LIN {X 0,Y 257.975,Z 573.967,A -85,B 0,C 180,E1 -19198.916,E2 -19198.916} C_VEL
LIN {X 0,Y 261.69,Z 562.431,A -85,B 0,C 180,E1 -19200.904,E2 -19200.904} C_VEL
LIN {X 0,Y 265.113,Z 550.939,A -85,B 0,C 180,E1 -19202.465,E2 -19202.465} C_VEL
LIN {X 0,Y 268.237,Z 538.403,A -85,B 0,C 180,E1 -19203.83,E2 -19203.83} C_VEL
LIN {X 0,Y 271.089,Z 525.455,A -85,B 0,C 180,E1 -19204.886,E2 -19204.886} C_VEL
LIN {X 0,Y 273.137,Z 513.119,A -85,B 0,C 180,E1 -19205.657,E2 -19205.657} C_VEL
LIN {X 0,Y 274.903,Z 498.669,A -85,B 0,C 180,E1 -19206.281,E2 -19206.281} C_VEL
LIN {X 0,Y 276.815,Z 466.117,A -85,B 0,C 180,E1 -19207.149,E2 -19207.149} C_VEL
LIN {X 0,Y 279.015,Z 421.953,A -85,B 0,C 180,E1 -19208.302,E2 -19208.302} C_VEL
LIN {X 0,Y 278.053,Z 415.902,A -85,B 0,C 180,E1 -19208.716,E2 -19208.716} C_VEL
LIN {X 0,Y 271.984,Z 402.227,A -85,B 0,C 180,E1 -19210.518,E2 -19210.518} C_VEL
LIN {X 0,Y 265.036,Z 388.919,A -85,B 0,C 180,E1 -19212.665,E2 -19212.665} C_VEL
LIN {X 0,Y 258.695,Z 378.17,A -85,B 0,C 180,E1 -19214.774,E2 -19214.774} C_VEL
LIN {X 0,Y 255.82,Z 373.588,A -85,B 0,C 180,E1 -19215.796,E2 -19215.796} C_VEL
LIN {X 0,Y 252.154,Z 368.029,A -85,B 0,C 180,E1 -19217.157,E2 -19217.157} C_VEL
LIN {X 0,Y 248.387,Z 362.468,A -85,B 0,C 180,E1 -19218.642,E2 -19218.642} C_VEL
LIN {X 0,Y 245.206,Z 357.875,A -85,B 0,C 180,E1 -19219.976,E2 -19219.976} C_VEL
LIN {X 0,Y 244.693,Z 356.869,A -85,B 0,C 180,E1 -19220.278,E2 -19220.278} C_VEL
LIN {X 0,Y 242.615,Z 351.052,A -85,B 0,C 180,E1 -19224.2,E2 -19224.2} C_VEL
LIN {X 0,Y 242.003,Z 348.966,A -85,B 0,C 180,E1 -19225.759,E2 -19225.759} C_VEL
LIN {X 0,Y 242.032,Z 348.953,A -85,B 0,C 180,E1 -19230.586,E2 -19230.586} C_VEL
LIN {X 0,Y 242.062,Z 348.949,A -85,B 0,C 180,E1 -19234.182,E2 -19234.182} C_VEL
LIN {X 0,Y 242.047,Z 348.954,A -85,B 0,C 180,E1 -19238.296,E2 -19238.296} C_VEL
LIN {X 0,Y 242.157,Z 348.946,A -85,B 0,C 180,E1 -19243.277,E2 -19243.277} C_VEL
LIN {X 0,Y 242.18,Z 348.932,A -85,B 0,C 180,E1 -19248.279,E2 -19248.279} C_VEL
LIN {X 0,Y 242.428,Z 348.909,A -85,B 0,C 180,E1 -19251.665,E2 -19251.665} C_VEL
LIN {X 0,Y 242.237,Z 348.937,A -85,B 0,C 180,E1 -19255.006,E2 -19255.006} C_VEL
LIN {X 0,Y 242.615,Z 348.882,A -85,B 0,C 180,E1 -19258.339,E2 -19258.339} C_VEL
LIN {X 0,Y 242.611,Z 348.878,A -85,B 0,C 180,E1 -19261.659,E2 -19261.659} C_VEL
LIN {X 0,Y 242.388,Z 348.915,A -85,B 0,C 180,E1 -19266.66,E2 -19266.66} C_VEL
LIN {X 0,Y 242.258,Z 348.927,A -85,B 0,C 180,E1 -19270.023,E2 -19270.023} C_VEL
LIN {X 0,Y 242.118,Z 348.946,A -85,B 0,C 180,E1 -19275.143,E2 -19275.143} C_VEL
LIN {X 0,Y 242.033,Z 348.956,A -85,B 0,C 180,E1 -19278.627,E2 -19278.627} C_VEL
LIN {X 0,Y 242.051,Z 349.148,A -85,B 0,C 180,E1 -19280.941,E2 -19280.941} C_VEL
LIN {X 0,Y 242.928,Z 351.572,A -85,B 0,C 180,E1 -19281.413,E2 -19281.413} C_VEL
LIN {X 0,Y 244.626,Z 353.64,A -85,B 0,C 180,E1 -19282.152,E2 -19282.152} C_VEL
LIN {X 0,Y 246.198,Z 354.858,A -85,B 0,C 180,E1 -19282.777,E2 -19282.777} C_VEL
LIN {X 0,Y 247.972,Z 357.809,A -85,B 0,C 180,E1 -19283.543,E2 -19283.543} C_VEL
LIN {X 0,Y 250.246,Z 360.174,A -85,B 0,C 180,E1 -19284.416,E2 -19284.416} C_VEL
LIN {X 0,Y 252.657,Z 363.577,A -85,B 0,C 180,E1 -19285.344,E2 -19285.344} C_VEL
LIN {X 0,Y 254.065,Z 365.243,A -85,B 0,C 180,E1 -19285.854,E2 -19285.854} C_VEL
LIN {X 0,Y 257.823,Z 370.434,A -85,B 0,C 180,E1 -19287.194,E2 -19287.194} C_VEL
LIN {X 0,Y 263.731,Z 378.79,A -85,B 0,C 180,E1 -19289.154,E2 -19289.154} C_VEL
LIN {X 0,Y 268.187,Z 385.843,A -85,B 0,C 180,E1 -19290.532,E2 -19290.532} C_VEL
LIN {X 0,Y 274.772,Z 397.82,A -85,B 0,C 180,E1 -19292.488,E2 -19292.488} C_VEL
LIN {X 0,Y 279.803,Z 408.378,A -85,B 0,C 180,E1 -19293.928,E2 -19293.928} C_VEL
LIN {X 0,Y 275.706,Z 481.995,A -85,B 0,C 180,E1 -19295.821,E2 -19295.821} C_VEL
LIN {X 0,Y 274.177,Z 496.417,A -85,B 0,C 180,E1 -19296.459,E2 -19296.459} C_VEL
LIN {X 0,Y 271.973,Z 510.678,A -85,B 0,C 180,E1 -19297.385,E2 -19297.385} C_VEL
LIN {X 0,Y 269.519,Z 523.528,A -85,B 0,C 180,E1 -19298.533,E2 -19298.533} C_VEL
LIN {X 0,Y 266.589,Z 535.608,A -85,B 0,C 180,E1 -19299.895,E2 -19299.895} C_VEL
LIN {X 0,Y 263.53,Z 546.378,A -85,B 0,C 180,E1 -19301.407,E2 -19301.407} C_VEL
LIN {X 0,Y 259.867,Z 557.729,A -85,B 0,C 180,E1 -19303.382,E2 -19303.382} C_VEL
LIN {X 0,Y 256.225,Z 567.968,A -85,B 0,C 180,E1 -19305.616,E2 -19305.616} C_VEL
LIN {X 0,Y 252.654,Z 577.137,A -85,B 0,C 180,E1 -19308.12,E2 -19308.12} C_VEL
LIN {X 0,Y 249.548,Z 584.618,A -85,B 0,C 180,E1 -19310.681,E2 -19310.681} C_VEL
LIN {X 0,Y 246.917,Z 590.719,A -85,B 0,C 180,E1 -19313.295,E2 -19313.295} C_VEL
LIN {X 0,Y 244.315,Z 596.539,A -85,B 0,C 180,E1 -19316.533,E2 -19316.533} C_VEL
LIN {X 0,Y 242.516,Z 600.511,A -85,B 0,C 180,E1 -19319.528,E2 -19319.528} C_VEL
LIN {X 0,Y 241.298,Z 603.047,A -85,B 0,C 180,E1 -19322.226,E2 -19322.226} C_VEL
LIN {X 0,Y 240.472,Z 604.693,A -85,B 0,C 180,E1 -19324.957,E2 -19324.957} C_VEL
LIN {X 0,Y 239.921,Z 605.496,A -85,B 0,C 180,E1 -19327.618,E2 -19327.618} C_VEL
LIN {X 0,Y 239.591,Z 605.256,A -85,B 0,C 180,E1 -19331.178,E2 -19331.178} C_VEL
LIN {X 0,Y 239.637,Z 603.584,A -85,B 0,C 180,E1 -19334.697,E2 -19334.697} C_VEL
LIN {X 0,Y 240.013,Z 600.481,A -85,B 0,C 180,E1 -19338.174,E2 -19338.174} C_VEL
LIN {X 0,Y 240.569,Z 597.158,A -85,B 0,C 180,E1 -19340.755,E2 -19340.755} C_VEL
LIN {X 0,Y 241.354,Z 592.961,A -85,B 0,C 180,E1 -19343.313,E2 -19343.313} C_VEL
LIN {X 0,Y 242.308,Z 587.757,A -85,B 0,C 180,E1 -19345.843,E2 -19345.843} C_VEL
LIN {X 0,Y 243.892,Z 580.311,A -85,B 0,C 180,E1 -19348.763,E2 -19348.763} C_VEL
LIN {X 0,Y 245.618,Z 572.504,A -85,B 0,C 180,E1 -19351.231,E2 -19351.231} C_VEL
LIN {X 0,Y 247.632,Z 563.136,A -85,B 0,C 180,E1 -19353.663,E2 -19353.663} C_VEL
LIN {X 0,Y 249.825,Z 552.746,A -85,B 0,C 180,E1 -19355.854,E2 -19355.854} C_VEL
LIN {X 0,Y 252.095,Z 541.274,A -85,B 0,C 180,E1 -19357.812,E2 -19357.812} C_VEL
LIN {X 0,Y 254.36,Z 528.566,A -85,B 0,C 180,E1 -19359.544,E2 -19359.544} C_VEL
LIN {X 0,Y 256.247,Z 516.233,A -85,B 0,C 180,E1 -19360.87,E2 -19360.87} C_VEL
LIN {X 0,Y 257.878,Z 502.651,A -85,B 0,C 180,E1 -19361.995,E2 -19361.995} C_VEL
LIN {X 0,Y 259.068,Z 489.521,A -85,B 0,C 180,E1 -19362.785,E2 -19362.785} C_VEL
LIN {X 0,Y 259.965,Z 475.474,A -85,B 0,C 180,E1 -19363.334,E2 -19363.334} C_VEL
LIN {X 0,Y 263.004,Z 394.213,A -85,B 0,C 180,E1 -19365.519,E2 -19365.519} C_VEL
LIN {X 0,Y 255.473,Z 375.166,A -85,B 0,C 180,E1 -19367.04,E2 -19367.04} C_VEL
LIN {X 0,Y 248.343,Z 361.226,A -85,B 0,C 180,E1 -19368.445,E2 -19368.445} C_VEL
LIN {X 0,Y 243.171,Z 351.999,A -85,B 0,C 180,E1 -19369.494,E2 -19369.494} C_VEL
LIN {X 0,Y 242.129,Z 349.364,A -85,B 0,C 180,E1 -19369.74,E2 -19369.74} C_VEL
LIN {X 0,Y 242.068,Z 348.964,A -85,B 0,C 180,E1 -19369.773,E2 -19369.773} C_VEL
LIN {X 0,Y 242.024,Z 348.964,A -85,B 0,C 180,E1 -19373.989,E2 -19373.989} C_VEL
LIN {X 0,Y 241.96,Z 348.97,A -85,B 0,C 180,E1 -19377.695,E2 -19377.695} C_VEL
LIN {X 0,Y 241.948,Z 348.97,A -85,B 0,C 180,E1 -19381.525,E2 -19381.525} C_VEL
LIN {X 0,Y 241.978,Z 348.959,A -85,B 0,C 180,E1 -19385.589,E2 -19385.589} C_VEL
LIN {X 0,Y 241.94,Z 348.972,A -85,B 0,C 180,E1 -19389.724,E2 -19389.724} C_VEL
LIN {X 0,Y 241.897,Z 348.958,A -85,B 0,C 180,E1 -19394.212,E2 -19394.212} C_VEL
LIN {X 0,Y 241.906,Z 348.974,A -85,B 0,C 180,E1 -19398.072,E2 -19398.072} C_VEL
LIN {X 0,Y 241.966,Z 348.95,A -85,B 0,C 180,E1 -19402.415,E2 -19402.415} C_VEL
LIN {X 0,Y 241.98,Z 348.956,A -85,B 0,C 180,E1 -19406.508,E2 -19406.508} C_VEL
LIN {X 0,Y 241.973,Z 348.967,A -85,B 0,C 180,E1 -19410.617,E2 -19410.617} C_VEL
LIN {X 0,Y 241.998,Z 348.964,A -85,B 0,C 180,E1 -19414.198,E2 -19414.198} C_VEL
LIN {X 0,Y 241.988,Z 348.961,A -85,B 0,C 180,E1 -19418.339,E2 -19418.339} C_VEL
LIN {X 0,Y 242.109,Z 348.947,A -85,B 0,C 180,E1 -19423.325,E2 -19423.325} C_VEL
LIN {X 0,Y 242.157,Z 348.916,A -85,B 0,C 180,E1 -19428.279,E2 -19428.279} C_VEL
LIN {X 0,Y 242.372,Z 348.913,A -85,B 0,C 180,E1 -19431.664,E2 -19431.664} C_VEL
LIN {X 0,Y 242.402,Z 348.913,A -85,B 0,C 180,E1 -19433.341,E2 -19433.341} C_VEL
LIN {X 0,Y 242.629,Z 348.862,A -85,B 0,C 180,E1 -19438.341,E2 -19438.341} C_VEL
LIN {X 0,Y 242.628,Z 348.869,A -85,B 0,C 180,E1 -19441.66,E2 -19441.66} C_VEL
LIN {X 0,Y 242.412,Z 348.911,A -85,B 0,C 180,E1 -19446.66,E2 -19446.66} C_VEL
LIN {X 0,Y 242.38,Z 348.91,A -85,B 0,C 180,E1 -19447.995,E2 -19447.995} C_VEL
LIN {X 0,Y 242.071,Z 348.952,A -85,B 0,C 180,E1 -19448.921,E2 -19448.921} C_VEL
LIN {X 0,Y 240.681,Z 349.13,A -85,B 0,C 180,E1 -19450.286,E2 -19450.286} C_VEL
LIN {X 0,Y 236.209,Z 349.682,A -85,B 0,C 180,E1 -19453.469,E2 -19453.469} C_VEL
LIN {X 0,Y 235.168,Z 349.812,A -85,B 0,C 180,E1 -19454.899,E2 -19454.899} C_VEL
LIN {X 0,Y 235.106,Z 349.821,A -85,B 0,C 180,E1 -19455.383,E2 -19455.383} C_VEL
LIN {X 0,Y 235.015,Z 349.828,A -85,B 0,C 180,E1 -19459.206,E2 -19459.206} C_VEL
LIN {X 0,Y 234.968,Z 349.839,A -85,B 0,C 180,E1 -19462.883,E2 -19462.883} C_VEL
LIN {X 0,Y 234.974,Z 349.837,A -85,B 0,C 180,E1 -19466.657,E2 -19466.657} C_VEL
LIN {X 0,Y 234.928,Z 349.842,A -85,B 0,C 180,E1 -19470.569,E2 -19470.569} C_VEL
LIN {X 0,Y 234.936,Z 349.844,A -85,B 0,C 180,E1 -19474.638,E2 -19474.638} C_VEL
LIN {X 0,Y 234.947,Z 349.833,A -85,B 0,C 180,E1 -19478.944,E2 -19478.944} C_VEL
LIN {X 0,Y 234.895,Z 349.851,A -85,B 0,C 180,E1 -19483.485,E2 -19483.485} C_VEL
LIN {X 0,Y 234.911,Z 349.935,A -85,B 0,C 180,E1 -19487.578,E2 -19487.578} C_VEL
LIN {X 0,Y 237.393,Z 359.445,A -85,B 0,C 180,E1 -19491.38,E2 -19491.38} C_VEL
LIN {X 0,Y 245.889,Z 378.551,A -85,B 0,C 180,E1 -19493.277,E2 -19493.277} C_VEL
LIN {X 0,Y 252.992,Z 396.867,A -85,B 0,C 180,E1 -19494.823,E2 -19494.823} C_VEL
LIN {X 0,Y 256.061,Z 418.699,A -85,B 0,C 180,E1 -19495.906,E2 -19495.906} C_VEL
LIN {X 0,Y 252.882,Z 498.38,A -85,B 0,C 180,E1 -19498.125,E2 -19498.125} C_VEL
LIN {X 0,Y 251.642,Z 512.962,A -85,B 0,C 180,E1 -19498.831,E2 -19498.831} C_VEL
LIN {X 0,Y 249.936,Z 526.964,A -85,B 0,C 180,E1 -19499.824,E2 -19499.824} C_VEL
LIN {X 0,Y 248.041,Z 539.106,A -85,B 0,C 180,E1 -19500.972,E2 -19500.972} C_VEL
LIN {X 0,Y 245.689,Z 552.322,A -85,B 0,C 180,E1 -19502.589,E2 -19502.589} C_VEL
LIN {X 0,Y 243.884,Z 561.254,A -85,B 0,C 180,E1 -19503.929,E2 -19503.929} C_VEL
LIN {X 0,Y 241.535,Z 572.372,A -85,B 0,C 180,E1 -19505.959,E2 -19505.959} C_VEL
LIN {X 0,Y 239.411,Z 581.659,A -85,B 0,C 180,E1 -19508.019,E2 -19508.019} C_VEL
LIN {X 0,Y 237.353,Z 590.965,A -85,B 0,C 180,E1 -19510.541,E2 -19510.541} C_VEL
LIN {X 0,Y 235.71,Z 598.695,A -85,B 0,C 180,E1 -19513.098,E2 -19513.098} C_VEL
LIN {X 0,Y 234.339,Z 606.056,A -85,B 0,C 180,E1 -19516.116,E2 -19516.116} C_VEL
LIN {X 0,Y 233.452,Z 611.184,A -85,B 0,C 180,E1 -19518.714,E2 -19518.714} C_VEL
LIN {X 0,Y 232.936,Z 616.448,A -85,B 0,C 180,E1 -19522.195,E2 -19522.195} C_VEL
LIN {X 0,Y 232.781,Z 619.653,A -85,B 0,C 180,E1 -19525.088,E2 -19525.088} C_VEL
LIN {X 0,Y 232.859,Z 621.993,A -85,B 0,C 180,E1 -19528.269,E2 -19528.269} C_VEL
LIN {X 0,Y 232.89,Z 622.761,A -85,B 0,C 180,E1 -19529.998,E2 -19529.998} C_VEL
LIN {X 0,Y 232.815,Z 623.182,A -85,B 0,C 180,E1 -19531.728,E2 -19531.728} C_VEL
LIN {X 0,Y 232.729,Z 623.018,A -85,B 0,C 180,E1 -19535.196,E2 -19535.196} C_VEL
LIN {X 0,Y 233.035,Z 621.536,A -85,B 0,C 180,E1 -19538.671,E2 -19538.671} C_VEL
LIN {X 0,Y 233.862,Z 618.721,A -85,B 0,C 180,E1 -19542.142,E2 -19542.142} C_VEL
LIN {X 0,Y 235.558,Z 614.505,A -85,B 0,C 180,E1 -19545.574,E2 -19545.574} C_VEL
LIN {X 0,Y 237.772,Z 608.769,A -85,B 0,C 180,E1 -19548.972,E2 -19548.972} C_VEL
LIN {X 0,Y 240.51,Z 602.355,A -85,B 0,C 180,E1 -19551.872,E2 -19551.872} C_VEL
LIN {X 0,Y 243.889,Z 594.43,A -85,B 0,C 180,E1 -19554.696,E2 -19554.696} C_VEL
LIN {X 0,Y 247.294,Z 586.189,A -85,B 0,C 180,E1 -19557.045,E2 -19557.045} C_VEL
LIN {X 0,Y 251.175,Z 576.318,A -85,B 0,C 180,E1 -19559.316,E2 -19559.316} C_VEL
LIN {X 0,Y 254.896,Z 565.57,A -85,B 0,C 180,E1 -19561.323,E2 -19561.323} C_VEL
LIN {X 0,Y 258.787,Z 553.302,A -85,B 0,C 180,E1 -19563.128,E2 -19563.128} C_VEL
LIN {X 0,Y 262.027,Z 541.385,A -85,B 0,C 180,E1 -19564.512,E2 -19564.512} C_VEL
LIN {X 0,Y 265.344,Z 527.122,A -85,B 0,C 180,E1 -19565.755,E2 -19565.755} C_VEL
LIN {X 0,Y 267.827,Z 513.201,A -85,B 0,C 180,E1 -19566.652,E2 -19566.652} C_VEL
LIN {X 0,Y 269.641,Z 499.013,A -85,B 0,C 180,E1 -19567.277,E2 -19567.277} C_VEL
LIN {X 0,Y 271.203,Z 474.142,A -85,B 0,C 180,E1 -19567.97,E2 -19567.97} C_VEL
LIN {X 0,Y 273.906,Z 423.079,A -85,B 0,C 180,E1 -19569.31,E2 -19569.31} C_VEL
LIN {X 0,Y 273.254,Z 419.085,A -85,B 0,C 180,E1 -19569.598,E2 -19569.598} C_VEL
LIN {X 0,Y 267.285,Z 405.619,A -85,B 0,C 180,E1 -19571.453,E2 -19571.453} C_VEL
LIN {X 0,Y 260.86,Z 393.201,A -85,B 0,C 180,E1 -19573.536,E2 -19573.536} C_VEL
LIN {X 0,Y 255.254,Z 383.443,A -85,B 0,C 180,E1 -19575.509,E2 -19575.509} C_VEL
LIN {X 0,Y 252.276,Z 378.651,A -85,B 0,C 180,E1 -19576.612,E2 -19576.612} C_VEL
LIN {X 0,Y 248.97,Z 373.514,A -85,B 0,C 180,E1 -19577.895,E2 -19577.895} C_VEL
LIN {X 0,Y 245.215,Z 367.905,A -85,B 0,C 180,E1 -19579.44,E2 -19579.44} C_VEL
LIN {X 0,Y 242.099,Z 363.161,A -85,B 0,C 180,E1 -19580.816,E2 -19580.816} C_VEL
LIN {X 0,Y 237.776,Z 357.492,A -85,B 0,C 180,E1 -19582.851,E2 -19582.851} C_VEL
LIN {X 0,Y 237.187,Z 356.277,A -85,B 0,C 180,E1 -19583.248,E2 -19583.248} C_VEL
LIN {X 0,Y 235.514,Z 351.829,A -85,B 0,C 180,E1 -19586.67,E2 -19586.67} C_VEL
LIN {X 0,Y 234.938,Z 349.844,A -85,B 0,C 180,E1 -19588.432,E2 -19588.432} C_VEL
LIN {X 0,Y 234.947,Z 349.84,A -85,B 0,C 180,E1 -19591.405,E2 -19591.405} C_VEL
LIN {X 0,Y 234.982,Z 349.84,A -85,B 0,C 180,E1 -19595.246,E2 -19595.246} C_VEL
LIN {X 0,Y 235.005,Z 349.838,A -85,B 0,C 180,E1 -19598.969,E2 -19598.969} C_VEL
LIN {X 0,Y 235.09,Z 349.827,A -85,B 0,C 180,E1 -19603.058,E2 -19603.058} C_VEL
LIN {X 0,Y 235.14,Z 349.812,A -85,B 0,C 180,E1 -19607.923,E2 -19607.923} C_VEL
LIN {X 0,Y 235.383,Z 349.789,A -85,B 0,C 180,E1 -19611.414,E2 -19611.414} C_VEL
LIN {X 0,Y 235.396,Z 349.775,A -85,B 0,C 180,E1 -19613.141,E2 -19613.141} C_VEL
LIN {X 0,Y 235.574,Z 349.758,A -85,B 0,C 180,E1 -19618.29,E2 -19618.29} C_VEL
LIN {X 0,Y 235.57,Z 349.755,A -85,B 0,C 180,E1 -19621.709,E2 -19621.709} C_VEL
LIN {X 0,Y 235.339,Z 349.795,A -85,B 0,C 180,E1 -19626.86,E2 -19626.86} C_VEL
LIN {X 0,Y 235.204,Z 349.808,A -85,B 0,C 180,E1 -19630.327,E2 -19630.327} C_VEL
LIN {X 0,Y 235.066,Z 349.821,A -85,B 0,C 180,E1 -19635.609,E2 -19635.609} C_VEL
LIN {X 0,Y 234.986,Z 349.84,A -85,B 0,C 180,E1 -19638.02,E2 -19638.02} C_VEL
LIN {X 0,Y 235.756,Z 352.277,A -85,B 0,C 180,E1 -19638.521,E2 -19638.521} C_VEL
LIN {X 0,Y 237.564,Z 354.492,A -85,B 0,C 180,E1 -19639.439,E2 -19639.439} C_VEL
LIN {X 0,Y 239.331,Z 355.648,A -85,B 0,C 180,E1 -19640.24,E2 -19640.24} C_VEL
LIN {X 0,Y 241.267,Z 358.972,A -85,B 0,C 180,E1 -19641.2,E2 -19641.2} C_VEL
LIN {X 0,Y 243.595,Z 361.29,A -85,B 0,C 180,E1 -19642.195,E2 -19642.195} C_VEL
LIN {X 0,Y 246.202,Z 364.832,A -85,B 0,C 180,E1 -19643.304,E2 -19643.304} C_VEL
LIN {X 0,Y 247.587,Z 366.496,A -85,B 0,C 180,E1 -19643.859,E2 -19643.859} C_VEL
LIN {X 0,Y 250.513,Z 370.227,A -85,B 0,C 180,E1 -19644.995,E2 -19644.995} C_VEL
LIN {X 0,Y 257.73,Z 380.445,A -85,B 0,C 180,E1 -19647.617,E2 -19647.617} C_VEL
LIN {X 0,Y 262.95,Z 388.395,A -85,B 0,C 180,E1 -19649.358,E2 -19649.358} C_VEL
LIN {X 0,Y 269.193,Z 399.609,A -85,B 0,C 180,E1 -19651.315,E2 -19651.315} C_VEL
LIN {X 0,Y 274.616,Z 410.811,A -85,B 0,C 180,E1 -19652.944,E2 -19652.944} C_VEL
LIN {X 0,Y 270.472,Z 482.653,A -85,B 0,C 180,E1 -19654.823,E2 -19654.823} C_VEL
LIN {X 0,Y 268.878,Z 496.989,A -85,B 0,C 180,E1 -19655.469,E2 -19655.469} C_VEL
LIN {X 0,Y 266.708,Z 510.575,A -85,B 0,C 180,E1 -19656.359,E2 -19656.359} C_VEL
LIN {X 0,Y 264.302,Z 522.735,A -85,B 0,C 180,E1 -19657.436,E2 -19657.436} C_VEL
LIN {X 0,Y 260.961,Z 536.144,A -85,B 0,C 180,E1 -19658.958,E2 -19658.958} C_VEL
LIN {X 0,Y 257.63,Z 547.366,A -85,B 0,C 180,E1 -19660.57,E2 -19660.57} C_VEL
LIN {X 0,Y 253.896,Z 558.336,A -85,B 0,C 180,E1 -19662.527,E2 -19662.527} C_VEL
LIN {X 0,Y 250.209,Z 568.234,A -85,B 0,C 180,E1 -19664.738,E2 -19664.738} C_VEL
LIN {X 0,Y 246.481,Z 577.353,A -85,B 0,C 180,E1 -19667.278,E2 -19667.278} C_VEL
LIN {X 0,Y 243.092,Z 585.034,A -85,B 0,C 180,E1 -19669.966,E2 -19669.966} C_VEL
LIN {X 0,Y 240.738,Z 590.158,A -85,B 0,C 180,E1 -19672.191,E2 -19672.191} C_VEL
LIN {X 0,Y 238.365,Z 595.225,A -85,B 0,C 180,E1 -19674.907,E2 -19674.907} C_VEL
LIN {X 0,Y 236.437,Z 599.219,A -85,B 0,C 180,E1 -19677.655,E2 -19677.655} C_VEL
LIN {X 0,Y 234.562,Z 602.996,A -85,B 0,C 180,E1 -19681.356,E2 -19681.356} C_VEL
LIN {X 0,Y 233.348,Z 605.184,A -85,B 0,C 180,E1 -19685.063,E2 -19685.063} C_VEL
LIN {X 0,Y 232.652,Z 605.869,A -85,B 0,C 180,E1 -19688.748,E2 -19688.748} C_VEL
LIN {X 0,Y 232.449,Z 605.06,A -85,B 0,C 180,E1 -19692.403,E2 -19692.403} C_VEL
LIN {X 0,Y 232.659,Z 602.815,A -85,B 0,C 180,E1 -19696.017,E2 -19696.017} C_VEL
LIN {X 0,Y 233.219,Z 599.12,A -85,B 0,C 180,E1 -19699.585,E2 -19699.585} C_VEL
LIN {X 0,Y 234.162,Z 593.891,A -85,B 0,C 180,E1 -19703.106,E2 -19703.106} C_VEL
LIN {X 0,Y 235.148,Z 588.824,A -85,B 0,C 180,E1 -19705.717,E2 -19705.717} C_VEL
LIN {X 0,Y 236.711,Z 581.566,A -85,B 0,C 180,E1 -19708.726,E2 -19708.726} C_VEL
LIN {X 0,Y 238.44,Z 573.961,A -85,B 0,C 180,E1 -19711.268,E2 -19711.268} C_VEL
LIN {X 0,Y 240.522,Z 564.826,A -85,B 0,C 180,E1 -19713.771,E2 -19713.771} C_VEL
LIN {X 0,Y 242.942,Z 553.768,A -85,B 0,C 180,E1 -19716.229,E2 -19716.229} C_VEL
LIN {X 0,Y 245.297,Z 542.467,A -85,B 0,C 180,E1 -19718.238,E2 -19718.238} C_VEL
LIN {X 0,Y 247.621,Z 529.96,A -85,B 0,C 180,E1 -19720.013,E2 -19720.013} C_VEL
LIN {X 0,Y 249.541,Z 517.917,A -85,B 0,C 180,E1 -19721.372,E2 -19721.372} C_VEL
LIN {X 0,Y 251.23,Z 504.752,A -85,B 0,C 180,E1 -19722.523,E2 -19722.523} C_VEL
LIN {X 0,Y 252.6,Z 490.541,A -85,B 0,C 180,E1 -19723.425,E2 -19723.425} C_VEL
LIN {X 0,Y 253.526,Z 476.632,A -85,B 0,C 180,E1 -19723.998,E2 -19723.998} C_VEL
LIN {X 0,Y 256.678,Z 395.849,A -85,B 0,C 180,E1 -19726.222,E2 -19726.222} C_VEL
LIN {X 0,Y 249.425,Z 377.53,A -85,B 0,C 180,E1 -19727.752,E2 -19727.752} C_VEL
LIN {X 0,Y 241.597,Z 362.494,A -85,B 0,C 180,E1 -19729.358,E2 -19729.358} C_VEL
LIN {X 0,Y 236.399,Z 353.278,A -85,B 0,C 180,E1 -19730.468,E2 -19730.468} C_VEL
LIN {X 0,Y 235.172,Z 350.826,A -85,B 0,C 180,E1 -19730.749,E2 -19730.749} C_VEL
LIN {X 0,Y 234.976,Z 349.847,A -85,B 0,C 180,E1 -19730.847,E2 -19730.847} C_VEL
LIN {X 0,Y 234.953,Z 349.847,A -85,B 0,C 180,E1 -19734.759,E2 -19734.759} C_VEL
LIN {X 0,Y 234.896,Z 349.851,A -85,B 0,C 180,E1 -19738.603,E2 -19738.603} C_VEL
LIN {X 0,Y 234.94,Z 349.848,A -85,B 0,C 180,E1 -19743.115,E2 -19743.115} C_VEL
LIN {X 0,Y 234.915,Z 349.833,A -85,B 0,C 180,E1 -19746.753,E2 -19746.753} C_VEL
LIN {X 0,Y 234.913,Z 349.846,A -85,B 0,C 180,E1 -19748.937,E2 -19748.937} C_VEL
LIN {X 0,Y 234.853,Z 349.838,A -85,B 0,C 180,E1 -19753.495,E2 -19753.495} C_VEL
LIN {X 0,Y 234.853,Z 349.844,A -85,B 0,C 180,E1 -19756.507,E2 -19756.507} C_VEL
LIN {X 0,Y 234.92,Z 349.838,A -85,B 0,C 180,E1 -19761.08,E2 -19761.08} C_VEL
LIN {X 0,Y 234.924,Z 349.826,A -85,B 0,C 180,E1 -19765.362,E2 -19765.362} C_VEL
LIN {X 0,Y 234.897,Z 349.849,A -85,B 0,C 180,E1 -19769.428,E2 -19769.428} C_VEL
LIN {X 0,Y 234.942,Z 349.841,A -85,B 0,C 180,E1 -19773.822,E2 -19773.822} C_VEL
LIN {X 0,Y 234.939,Z 349.84,A -85,B 0,C 180,E1 -19778.964,E2 -19778.964} C_VEL
LIN {X 0,Y 235.053,Z 349.826,A -85,B 0,C 180,E1 -19783.099,E2 -19783.099} C_VEL
LIN {X 0,Y 235.089,Z 349.793,A -85,B 0,C 180,E1 -19787.921,E2 -19787.921} C_VEL
LIN {X 0,Y 235.309,Z 349.791,A -85,B 0,C 180,E1 -19791.412,E2 -19791.412} C_VEL
LIN {X 0,Y 235.353,Z 349.791,A -85,B 0,C 180,E1 -19793.14,E2 -19793.14} C_VEL
LIN {X 0,Y 235.588,Z 349.738,A -85,B 0,C 180,E1 -19798.291,E2 -19798.291} C_VEL
LIN {X 0,Y 235.586,Z 349.745,A -85,B 0,C 180,E1 -19801.71,E2 -19801.71} C_VEL
LIN {X 0,Y 235.363,Z 349.789,A -85,B 0,C 180,E1 -19806.86,E2 -19806.86} C_VEL
LIN {X 0,Y 235.219,Z 349.81,A -85,B 0,C 180,E1 -19810.328,E2 -19810.328} C_VEL
LIN {X 0,Y 235.106,Z 349.821,A -85,B 0,C 180,E1 -19815.383,E2 -19815.383} C_VEL
LIN {X 0,Y 234.828,Z 349.862,A -85,B 0,C 180,E1 -19816.339,E2 -19816.339} C_VEL
LIN {X 0,Y 233.491,Z 350.033,A -85,B 0,C 180,E1 -19817.749,E2 -19817.749} C_VEL
LIN {X 0,Y 229.083,Z 350.575,A -85,B 0,C 180,E1 -19821.038,E2 -19821.038} C_VEL
LIN {X 0,Y 228.002,Z 350.707,A -85,B 0,C 180,E1 -19822.514,E2 -19822.514} C_VEL
LIN {X 0,Y 227.913,Z 350.715,A -85,B 0,C 180,E1 -19823.016,E2 -19823.016} C_VEL
LIN {X 0,Y 227.948,Z 350.712,A -85,B 0,C 180,E1 -19826.602,E2 -19826.602} C_VEL
LIN {X 0,Y 227.903,Z 350.717,A -85,B 0,C 180,E1 -19830.291,E2 -19830.291} C_VEL
LIN {X 0,Y 227.883,Z 350.72,A -85,B 0,C 180,E1 -19833.72,E2 -19833.72} C_VEL
LIN {X 0,Y 227.849,Z 350.714,A -85,B 0,C 180,E1 -19838.091,E2 -19838.091} C_VEL
LIN {X 0,Y 227.818,Z 350.733,A -85,B 0,C 180,E1 -19842.741,E2 -19842.741} C_VEL
LIN {X 0,Y 227.871,Z 350.756,A -85,B 0,C 180,E1 -19846.709,E2 -19846.709} C_VEL
LIN {X 0,Y 230.078,Z 359.211,A -85,B 0,C 180,E1 -19850.212,E2 -19850.212} C_VEL
LIN {X 0,Y 237.802,Z 375.954,A -85,B 0,C 180,E1 -19852.032,E2 -19852.032} C_VEL
LIN {X 0,Y 245.687,Z 395.564,A -85,B 0,C 180,E1 -19853.825,E2 -19853.825} C_VEL
LIN {X 0,Y 247.388,Z 401.03,A -85,B 0,C 180,E1 -19854.236,E2 -19854.236} C_VEL
LIN {X 0,Y 249.792,Z 420.966,A -85,B 0,C 180,E1 -19855.21,E2 -19855.21} C_VEL
LIN {X 0,Y 246.538,Z 497.819,A -85,B 0,C 180,E1 -19857.386,E2 -19857.386} C_VEL
LIN {X 0,Y 245.28,Z 512.511,A -85,B 0,C 180,E1 -19858.109,E2 -19858.109} C_VEL
LIN {X 0,Y 243.434,Z 527.129,A -85,B 0,C 180,E1 -19859.172,E2 -19859.172} C_VEL
LIN {X 0,Y 241.489,Z 539.18,A -85,B 0,C 180,E1 -19860.345,E2 -19860.345} C_VEL
LIN {X 0,Y 239.117,Z 551.959,A -85,B 0,C 180,E1 -19861.947,E2 -19861.947} C_VEL
LIN {X 0,Y 237.198,Z 561.215,A -85,B 0,C 180,E1 -19863.374,E2 -19863.374} C_VEL
LIN {X 0,Y 234.984,Z 571.299,A -85,B 0,C 180,E1 -19865.245,E2 -19865.245} C_VEL
LIN {X 0,Y 232.751,Z 580.716,A -85,B 0,C 180,E1 -19867.355,E2 -19867.355} C_VEL
LIN {X 0,Y 230.579,Z 590.138,A -85,B 0,C 180,E1 -19869.945,E2 -19869.945} C_VEL
LIN {X 0,Y 228.794,Z 597.964,A -85,B 0,C 180,E1 -19872.571,E2 -19872.571} C_VEL
LIN {X 0,Y 227.754,Z 603.44,A -85,B 0,C 180,E1 -19874.792,E2 -19874.792} C_VEL
LIN {X 0,Y 226.672,Z 608.969,A -85,B 0,C 180,E1 -19877.463,E2 -19877.463} C_VEL
LIN {X 0,Y 225.966,Z 614.766,A -85,B 0,C 180,E1 -19881.052,E2 -19881.052} C_VEL
LIN {X 0,Y 225.731,Z 618.94,A -85,B 0,C 180,E1 -19884.639,E2 -19884.639} C_VEL
LIN {X 0,Y 225.767,Z 621.623,A -85,B 0,C 180,E1 -19888.215,E2 -19888.215} C_VEL
LIN {X 0,Y 225.822,Z 622.432,A -85,B 0,C 180,E1 -19889.998,E2 -19889.998} C_VEL
LIN {X 0,Y 225.724,Z 622.888,A -85,B 0,C 180,E1 -19891.783,E2 -19891.783} C_VEL
LIN {X 0,Y 225.643,Z 622.793,A -85,B 0,C 180,E1 -19895.36,E2 -19895.36} C_VEL
LIN {X 0,Y 225.98,Z 621.378,A -85,B 0,C 180,E1 -19898.944,E2 -19898.944} C_VEL
LIN {X 0,Y 226.874,Z 618.628,A -85,B 0,C 180,E1 -19902.522,E2 -19902.522} C_VEL
LIN {X 0,Y 228.675,Z 614.482,A -85,B 0,C 180,E1 -19906.056,E2 -19906.056} C_VEL
LIN {X 0,Y 231.035,Z 608.82,A -85,B 0,C 180,E1 -19909.547,E2 -19909.547} C_VEL
LIN {X 0,Y 233.906,Z 602.499,A -85,B 0,C 180,E1 -19912.523,E2 -19912.523} C_VEL
LIN {X 0,Y 237.468,Z 594.682,A -85,B 0,C 180,E1 -19915.411,E2 -19915.411} C_VEL
LIN {X 0,Y 241.01,Z 586.561,A -85,B 0,C 180,E1 -19917.81,E2 -19917.81} C_VEL
LIN {X 0,Y 245.037,Z 576.817,A -85,B 0,C 180,E1 -19920.125,E2 -19920.125} C_VEL
LIN {X 0,Y 248.869,Z 566.325,A -85,B 0,C 180,E1 -19922.147,E2 -19922.147} C_VEL
LIN {X 0,Y 252.928,Z 554.165,A -85,B 0,C 180,E1 -19923.999,E2 -19923.999} C_VEL
LIN {X 0,Y 256.277,Z 542.507,A -85,B 0,C 180,E1 -19925.401,E2 -19925.401} C_VEL
LIN {X 0,Y 259.685,Z 528.781,A -85,B 0,C 180,E1 -19926.66,E2 -19926.66} C_VEL
LIN {X 0,Y 262.341,Z 514.786,A -85,B 0,C 180,E1 -19927.609,E2 -19927.609} C_VEL
LIN {X 0,Y 264.322,Z 500.971,A -85,B 0,C 180,E1 -19928.248,E2 -19928.248} C_VEL
LIN {X 0,Y 265.522,Z 484.637,A -85,B 0,C 180,E1 -19928.758,E2 -19928.758} C_VEL
LIN {X 0,Y 268.892,Z 424.325,A -85,B 0,C 180,E1 -19930.349,E2 -19930.349} C_VEL
LIN {X 0,Y 268.448,Z 422.19,A -85,B 0,C 180,E1 -19930.532,E2 -19930.532} C_VEL
LIN {X 0,Y 263.147,Z 410.06,A -85,B 0,C 180,E1 -19932.258,E2 -19932.258} C_VEL
LIN {X 0,Y 257.365,Z 398.534,A -85,B 0,C 180,E1 -19934.237,E2 -19934.237} C_VEL
LIN {X 0,Y 251.795,Z 388.65,A -85,B 0,C 180,E1 -19936.285,E2 -19936.285} C_VEL
LIN {X 0,Y 248.768,Z 383.692,A -85,B 0,C 180,E1 -19937.458,E2 -19937.458} C_VEL
LIN {X 0,Y 245.731,Z 378.863,A -85,B 0,C 180,E1 -19938.692,E2 -19938.692} C_VEL
LIN {X 0,Y 242.549,Z 373.954,A -85,B 0,C 180,E1 -19940.059,E2 -19940.059} C_VEL
LIN {X 0,Y 238.735,Z 368.32,A -85,B 0,C 180,E1 -19941.814,E2 -19941.814} C_VEL
LIN {X 0,Y 234.832,Z 362.701,A -85,B 0,C 180,E1 -19943.787,E2 -19943.787} C_VEL
LIN {X 0,Y 230.823,Z 357.683,A -85,B 0,C 180,E1 -19945.975,E2 -19945.975} C_VEL
LIN {X 0,Y 229.562,Z 355.652,A -85,B 0,C 180,E1 -19946.822,E2 -19946.822} C_VEL
LIN {X 0,Y 228.94,Z 353.614,A -85,B 0,C 180,E1 -19948.542,E2 -19948.542} C_VEL
LIN {X 0,Y 227.92,Z 350.715,A -85,B 0,C 180,E1 -19951.448,E2 -19951.448} C_VEL
LIN {X 0,Y 227.923,Z 350.711,A -85,B 0,C 180,E1 -19954.425,E2 -19954.425} C_VEL
LIN {X 0,Y 227.956,Z 350.708,A -85,B 0,C 180,E1 -19958.286,E2 -19958.286} C_VEL
LIN {X 0,Y 228.029,Z 350.707,A -85,B 0,C 180,E1 -19962.825,E2 -19962.825} C_VEL
LIN {X 0,Y 228.087,Z 350.694,A -85,B 0,C 180,E1 -19967.543,E2 -19967.543} C_VEL
LIN {X 0,Y 228.319,Z 350.671,A -85,B 0,C 180,E1 -19971.146,E2 -19971.146} C_VEL
LIN {X 0,Y 228.349,Z 350.653,A -85,B 0,C 180,E1 -19972.928,E2 -19972.928} C_VEL
LIN {X 0,Y 228.532,Z 350.634,A -85,B 0,C 180,E1 -19978.237,E2 -19978.237} C_VEL
LIN {X 0,Y 228.528,Z 350.632,A -85,B 0,C 180,E1 -19981.762,E2 -19981.762} C_VEL
LIN {X 0,Y 228.292,Z 350.674,A -85,B 0,C 180,E1 -19987.073,E2 -19987.073} C_VEL
LIN {X 0,Y 228.134,Z 350.692,A -85,B 0,C 180,E1 -19990.651,E2 -19990.651} C_VEL
LIN {X 0,Y 228.017,Z 350.708,A -85,B 0,C 180,E1 -19994.616,E2 -19994.616} C_VEL
LIN {X 0,Y 228.732,Z 353.068,A -85,B 0,C 180,E1 -19995.196,E2 -19995.196} C_VEL
LIN {X 0,Y 230.597,Z 355.346,A -85,B 0,C 180,E1 -19996.312,E2 -19996.312} C_VEL
LIN {X 0,Y 232.624,Z 356.805,A -85,B 0,C 180,E1 -19997.391,E2 -19997.391} C_VEL
LIN {X 0,Y 234.402,Z 359.883,A -85,B 0,C 180,E1 -19998.406,E2 -19998.406} C_VEL
LIN {X 0,Y 237.06,Z 362.353,A -85,B 0,C 180,E1 -19999.707,E2 -19999.707} C_VEL
LIN {X 0,Y 239.281,Z 365.656,A -85,B 0,C 180,E1 -20000.809,E2 -20000.809} C_VEL
LIN {X 0,Y 241.024,Z 367.521,A -85,B 0,C 180,E1 -20001.591,E2 -20001.591} C_VEL
LIN {X 0,Y 243.922,Z 371.266,A -85,B 0,C 180,E1 -20002.85,E2 -20002.85} C_VEL
LIN {X 0,Y 248.928,Z 378.091,A -85,B 0,C 180,E1 -20004.877,E2 -20004.877} C_VEL
LIN {X 0,Y 254.329,Z 385.76,A -85,B 0,C 180,E1 -20006.89,E2 -20006.89} C_VEL
LIN {X 0,Y 259.75,Z 394.201,A -85,B 0,C 180,E1 -20008.777,E2 -20008.777} C_VEL
LIN {X 0,Y 265.644,Z 405.253,A -85,B 0,C 180,E1 -20010.712,E2 -20010.712} C_VEL
LIN {X 0,Y 269.557,Z 413.698,A -85,B 0,C 180,E1 -20011.95,E2 -20011.95} C_VEL
LIN {X 0,Y 265.365,Z 482.897,A -85,B 0,C 180,E1 -20013.771,E2 -20013.771} C_VEL
LIN {X 0,Y 263.649,Z 497.663,A -85,B 0,C 180,E1 -20014.446,E2 -20014.446} C_VEL
LIN {X 0,Y 261.312,Z 511.696,A -85,B 0,C 180,E1 -20015.39,E2 -20015.39} C_VEL
LIN {X 0,Y 258.869,Z 523.355,A -85,B 0,C 180,E1 -20016.443,E2 -20016.443} C_VEL
LIN {X 0,Y 255.779,Z 535.415,A -85,B 0,C 180,E1 -20017.821,E2 -20017.821} C_VEL
LIN {X 0,Y 252.212,Z 547.052,A -85,B 0,C 180,E1 -20019.486,E2 -20019.486} C_VEL
LIN {X 0,Y 248.382,Z 557.92,A -85,B 0,C 180,E1 -20021.428,E2 -20021.428} C_VEL
LIN {X 0,Y 244.567,Z 567.684,A -85,B 0,C 180,E1 -20023.604,E2 -20023.604} C_VEL
LIN {X 0,Y 240.759,Z 576.699,A -85,B 0,C 180,E1 -20026.112,E2 -20026.112} C_VEL
LIN {X 0,Y 237.223,Z 584.34,A -85,B 0,C 180,E1 -20028.765,E2 -20028.765} C_VEL
LIN {X 0,Y 233.676,Z 591.665,A -85,B 0,C 180,E1 -20032.03,E2 -20032.03} C_VEL
LIN {X 0,Y 230.934,Z 597.11,A -85,B 0,C 180,E1 -20035.253,E2 -20035.253} C_VEL
LIN {X 0,Y 228.828,Z 601.185,A -85,B 0,C 180,E1 -20038.528,E2 -20038.528} C_VEL
LIN {X 0,Y 227.059,Z 604.307,A -85,B 0,C 180,E1 -20042.338,E2 -20042.338} C_VEL
LIN {X 0,Y 225.969,Z 605.886,A -85,B 0,C 180,E1 -20046.153,E2 -20046.153} C_VEL
LIN {X 0,Y 225.468,Z 605.988,A -85,B 0,C 180,E1 -20049.95,E2 -20049.95} C_VEL
LIN {X 0,Y 225.378,Z 604.642,A -85,B 0,C 180,E1 -20053.703,E2 -20053.703} C_VEL
LIN {X 0,Y 225.516,Z 603.413,A -85,B 0,C 180,E1 -20055.565,E2 -20055.565} C_VEL
LIN {X 0,Y 226.046,Z 599.862,A -85,B 0,C 180,E1 -20059.25,E2 -20059.25} C_VEL
LIN {X 0,Y 226.835,Z 595.413,A -85,B 0,C 180,E1 -20062.498,E2 -20062.498} C_VEL
LIN {X 0,Y 227.993,Z 589.875,A -85,B 0,C 180,E1 -20065.582,E2 -20065.582} C_VEL
LIN {X 0,Y 229.515,Z 582.803,A -85,B 0,C 180,E1 -20068.686,E2 -20068.686} C_VEL
LIN {X 0,Y 231.61,Z 574.027,A -85,B 0,C 180,E1 -20071.74,E2 -20071.74} C_VEL
LIN {X 0,Y 233.758,Z 564.856,A -85,B 0,C 180,E1 -20074.312,E2 -20074.312} C_VEL
LIN {X 0,Y 236.287,Z 553.739,A -85,B 0,C 180,E1 -20076.834,E2 -20076.834} C_VEL
LIN {X 0,Y 238.731,Z 542.358,A -85,B 0,C 180,E1 -20078.892,E2 -20078.892} C_VEL
LIN {X 0,Y 241.174,Z 529.754,A -85,B 0,C 180,E1 -20080.708,E2 -20080.708} C_VEL
LIN {X 0,Y 243.158,Z 517.596,A -85,B 0,C 180,E1 -20082.097,E2 -20082.097} C_VEL
LIN {X 0,Y 244.908,Z 504.257,A -85,B 0,C 180,E1 -20083.273,E2 -20083.273} C_VEL
LIN {X 0,Y 246.276,Z 490.276,A -85,B 0,C 180,E1 -20084.168,E2 -20084.168} C_VEL
LIN {X 0,Y 247.272,Z 475.619,A -85,B 0,C 180,E1 -20084.765,E2 -20084.765} C_VEL
LIN {X 0,Y 250.414,Z 397.611,A -85,B 0,C 180,E1 -20086.953,E2 -20086.953} C_VEL
LIN {X 0,Y 243.868,Z 380.97,A -85,B 0,C 180,E1 -20088.393,E2 -20088.393} C_VEL
LIN {X 0,Y 236.613,Z 366.925,A -85,B 0,C 180,E1 -20089.94,E2 -20089.94} C_VEL
LIN {X 0,Y 229.35,Z 354.136,A -85,B 0,C 180,E1 -20091.565,E2 -20091.565} C_VEL
LIN {X 0,Y 228.091,Z 351.55,A -85,B 0,C 180,E1 -20091.874,E2 -20091.874} C_VEL
LIN {X 0,Y 227.942,Z 350.722,A -85,B 0,C 180,E1 -20091.955,E2 -20091.955} C_VEL
LIN {X 0,Y 227.921,Z 350.721,A -85,B 0,C 180,E1 -20096.593,E2 -20096.593} C_VEL
LIN {X 0,Y 227.87,Z 350.726,A -85,B 0,C 180,E1 -20100.281,E2 -20100.281} C_VEL
LIN {X 0,Y 227.877,Z 350.725,A -85,B 0,C 180,E1 -20103.722,E2 -20103.722} C_VEL
LIN {X 0,Y 227.841,Z 350.721,A -85,B 0,C 180,E1 -20108.093,E2 -20108.093} C_VEL
LIN {X 0,Y 227.786,Z 350.722,A -85,B 0,C 180,E1 -20112.75,E2 -20112.75} C_VEL
LIN {X 0,Y 227.81,Z 350.712,A -85,B 0,C 180,E1 -20115.2,E2 -20115.2} C_VEL
LIN {X 0,Y 227.799,Z 350.731,A -85,B 0,C 180,E1 -20119.618,E2 -20119.618} C_VEL
LIN {X 0,Y 227.863,Z 350.695,A -85,B 0,C 180,E1 -20124.126,E2 -20124.126} C_VEL
LIN {X 0,Y 227.856,Z 350.725,A -85,B 0,C 180,E1 -20128.376,E2 -20128.376} C_VEL
LIN {X 0,Y 227.843,Z 350.722,A -85,B 0,C 180,E1 -20132.44,E2 -20132.44} C_VEL
LIN {X 0,Y 227.868,Z 350.725,A -85,B 0,C 180,E1 -20136.363,E2 -20136.363} C_VEL
LIN {X 0,Y 227.892,Z 350.72,A -85,B 0,C 180,E1 -20140.171,E2 -20140.171} C_VEL
LIN {X 0,Y 228.003,Z 350.7,A -85,B 0,C 180,E1 -20143.895,E2 -20143.895} C_VEL
LIN {X 0,Y 228.129,Z 350.672,A -85,B 0,C 180,E1 -20149.349,E2 -20149.349} C_VEL
LIN {X 0,Y 228.304,Z 350.669,A -85,B 0,C 180,E1 -20152.928,E2 -20152.928} C_VEL
LIN {X 0,Y 228.546,Z 350.614,A -85,B 0,C 180,E1 -20158.238,E2 -20158.238} C_VEL
LIN {X 0,Y 228.544,Z 350.622,A -85,B 0,C 180,E1 -20161.763,E2 -20161.763} C_VEL
LIN {X 0,Y 228.315,Z 350.667,A -85,B 0,C 180,E1 -20167.073,E2 -20167.073} C_VEL
LIN {X 0,Y 228.15,Z 350.689,A -85,B 0,C 180,E1 -20170.652,E2 -20170.652} C_VEL
LIN {X 0,Y 228.037,Z 350.699,A -85,B 0,C 180,E1 -20175.388,E2 -20175.388} C_VEL
LIN {X 0,Y 228.009,Z 350.704,A -85,B 0,C 180,E1 -20177.953,E2 -20177.953} C_VEL
LIN {X 0,Y 227.937,Z 350.715,A -85,B 0,C 180,E1 -20182.33,E2 -20182.33} C_VEL
LIN {X 0,Y 227.913,Z 350.715,A -85,B 0,C 180,E1 -20183.016,E2 -20183.016} C_VEL
LIN {X 0,Y 227.256,Z 350.797,A -85,B 0,C 180,E1 -20184.49,E2 -20184.49} C_VEL
LIN {X 0,Y 224.448,Z 351.153,A -85,B 0,C 180,E1 -20186.898,E2 -20186.898} C_VEL
LIN {X 0,Y 221.198,Z 351.557,A -85,B 0,C 180,E1 -20189.872,E2 -20189.872} C_VEL
LIN {X 0,Y 220.834,Z 351.597,A -85,B 0,C 180,E1 -20190.902,E2 -20190.902} C_VEL
LIN {X 0,Y 220.807,Z 351.605,A -85,B 0,C 180,E1 -20194.955,E2 -20194.955} C_VEL
LIN {X 0,Y 220.812,Z 351.598,A -85,B 0,C 180,E1 -20199.536,E2 -20199.536} C_VEL
LIN {X 0,Y 220.781,Z 351.608,A -85,B 0,C 180,E1 -20204.453,E2 -20204.453} C_VEL
LIN {X 0,Y 220.811,Z 351.628,A -85,B 0,C 180,E1 -20205.808,E2 -20205.808} C_VEL
LIN {X 0,Y 222.692,Z 358.743,A -85,B 0,C 180,E1 -20208.933,E2 -20208.933} C_VEL
LIN {X 0,Y 231.088,Z 376.578,A -85,B 0,C 180,E1 -20211.026,E2 -20211.026} C_VEL
LIN {X 0,Y 238.448,Z 394.605,A -85,B 0,C 180,E1 -20212.786,E2 -20212.786} C_VEL
LIN {X 0,Y 241.37,Z 403.108,A -85,B 0,C 180,E1 -20213.494,E2 -20213.494} C_VEL
LIN {X 0,Y 243.585,Z 420.654,A -85,B 0,C 180,E1 -20214.395,E2 -20214.395} C_VEL
LIN {X 0,Y 240.261,Z 497.254,A -85,B 0,C 180,E1 -20216.611,E2 -20216.611} C_VEL
LIN {X 0,Y 239.033,Z 511.286,A -85,B 0,C 180,E1 -20217.297,E2 -20217.297} C_VEL
LIN {X 0,Y 237.284,Z 525.007,A -85,B 0,C 180,E1 -20218.281,E2 -20218.281} C_VEL
LIN {X 0,Y 235.234,Z 537.451,A -85,B 0,C 180,E1 -20219.474,E2 -20219.474} C_VEL
LIN {X 0,Y 232.813,Z 550.521,A -85,B 0,C 180,E1 -20221.117,E2 -20221.117} C_VEL
LIN {X 0,Y 230.853,Z 560.047,A -85,B 0,C 180,E1 -20222.593,E2 -20222.593} C_VEL
LIN {X 0,Y 228.252,Z 571.223,A -85,B 0,C 180,E1 -20224.707,E2 -20224.707} C_VEL
LIN {X 0,Y 225.723,Z 581.438,A -85,B 0,C 180,E1 -20227.094,E2 -20227.094} C_VEL
LIN {X 0,Y 223.514,Z 590.693,A -85,B 0,C 180,E1 -20229.763,E2 -20229.763} C_VEL
LIN {X 0,Y 221.549,Z 599.525,A -85,B 0,C 180,E1 -20232.935,E2 -20232.935} C_VEL
LIN {X 0,Y 220.07,Z 606.623,A -85,B 0,C 180,E1 -20236.141,E2 -20236.141} C_VEL
LIN {X 0,Y 219.21,Z 611.519,A -85,B 0,C 180,E1 -20238.908,E2 -20238.908} C_VEL
LIN {X 0,Y 218.801,Z 615.48,A -85,B 0,C 180,E1 -20241.688,E2 -20241.688} C_VEL
LIN {X 0,Y 218.594,Z 619.271,A -85,B 0,C 180,E1 -20245.335,E2 -20245.335} C_VEL
LIN {X 0,Y 218.678,Z 621.24,A -85,B 0,C 180,E1 -20248.157,E2 -20248.157} C_VEL
LIN {X 0,Y 218.754,Z 622.085,A -85,B 0,C 180,E1 -20249.998,E2 -20249.998} C_VEL
LIN {X 0,Y 218.635,Z 622.575,A -85,B 0,C 180,E1 -20251.84,E2 -20251.84} C_VEL
LIN {X 0,Y 218.564,Z 622.551,A -85,B 0,C 180,E1 -20255.534,E2 -20255.534} C_VEL
LIN {X 0,Y 218.943,Z 621.209,A -85,B 0,C 180,E1 -20259.234,E2 -20259.234} C_VEL
LIN {X 0,Y 219.899,Z 618.536,A -85,B 0,C 180,E1 -20262.926,E2 -20262.926} C_VEL
LIN {X 0,Y 221.797,Z 614.47,A -85,B 0,C 180,E1 -20266.568,E2 -20266.568} C_VEL
LIN {X 0,Y 224.327,Z 608.899,A -85,B 0,C 180,E1 -20270.157,E2 -20270.157} C_VEL
LIN {X 0,Y 227.346,Z 602.666,A -85,B 0,C 180,E1 -20273.211,E2 -20273.211} C_VEL
LIN {X 0,Y 231.084,Z 594.945,A -85,B 0,C 180,E1 -20276.165,E2 -20276.165} C_VEL
LIN {X 0,Y 234.771,Z 586.933,A -85,B 0,C 180,E1 -20278.616,E2 -20278.616} C_VEL
LIN {X 0,Y 238.949,Z 577.316,A -85,B 0,C 180,E1 -20280.976,E2 -20280.976} C_VEL
LIN {X 0,Y 242.878,Z 567.098,A -85,B 0,C 180,E1 -20283.011,E2 -20283.011} C_VEL
LIN {X 0,Y 247.116,Z 555.006,A -85,B 0,C 180,E1 -20284.913,E2 -20284.913} C_VEL
LIN {X 0,Y 251.019,Z 542.034,A -85,B 0,C 180,E1 -20286.507,E2 -20286.507} C_VEL
LIN {X 0,Y 254.337,Z 529.268,A -85,B 0,C 180,E1 -20287.687,E2 -20287.687} C_VEL
LIN {X 0,Y 257.201,Z 514.866,A -85,B 0,C 180,E1 -20288.684,E2 -20288.684} C_VEL
LIN {X 0,Y 259.286,Z 500.68,A -85,B 0,C 180,E1 -20289.35,E2 -20289.35} C_VEL
LIN {X 0,Y 260.617,Z 483.023,A -85,B 0,C 180,E1 -20289.898,E2 -20289.898} C_VEL
LIN {X 0,Y 263.939,Z 425.816,A -85,B 0,C 180,E1 -20291.425,E2 -20291.425} C_VEL
LIN {X 0,Y 258.927,Z 414.178,A -85,B 0,C 180,E1 -20293.137,E2 -20293.137} C_VEL
LIN {X 0,Y 253.026,Z 402.162,A -85,B 0,C 180,E1 -20295.29,E2 -20295.29} C_VEL
LIN {X 0,Y 246.816,Z 390.969,A -85,B 0,C 180,E1 -20297.724,E2 -20297.724} C_VEL
LIN {X 0,Y 241.945,Z 383.315,A -85,B 0,C 180,E1 -20299.769,E2 -20299.769} C_VEL
LIN {X 0,Y 239.308,Z 379.177,A -85,B 0,C 180,E1 -20300.965,E2 -20300.965} C_VEL
LIN {X 0,Y 235.837,Z 373.874,A -85,B 0,C 180,E1 -20302.664,E2 -20302.664} C_VEL
LIN {X 0,Y 231.779,Z 368.006,A -85,B 0,C 180,E1 -20304.821,E2 -20304.821} C_VEL
LIN {X 0,Y 228.253,Z 363.338,A -85,B 0,C 180,E1 -20306.87,E2 -20306.87} C_VEL
LIN {X 0,Y 226.918,Z 361.546,A -85,B 0,C 180,E1 -20307.706,E2 -20307.706} C_VEL
LIN {X 0,Y 222.742,Z 356.303,A -85,B 0,C 180,E1 -20310.591,E2 -20310.591} C_VEL
LIN {X 0,Y 222.111,Z 355.018,A -85,B 0,C 180,E1 -20311.148,E2 -20311.148} C_VEL
LIN {X 0,Y 220.855,Z 351.597,A -85,B 0,C 180,E1 -20315.061,E2 -20315.061} C_VEL
LIN {X 0,Y 220.887,Z 351.593,A -85,B 0,C 180,E1 -20319.513,E2 -20319.513} C_VEL
LIN {X 0,Y 221.01,Z 351.577,A -85,B 0,C 180,E1 -20323.369,E2 -20323.369} C_VEL
LIN {X 0,Y 221.11,Z 351.554,A -85,B 0,C 180,E1 -20329.005,E2 -20329.005} C_VEL
LIN {X 0,Y 221.287,Z 351.533,A -85,B 0,C 180,E1 -20332.701,E2 -20332.701} C_VEL
LIN {X 0,Y 221.466,Z 351.514,A -85,B 0,C 180,E1 -20338.181,E2 -20338.181} C_VEL
LIN {X 0,Y 221.462,Z 351.512,A -85,B 0,C 180,E1 -20341.818,E2 -20341.818} C_VEL
LIN {X 0,Y 221.23,Z 351.554,A -85,B 0,C 180,E1 -20347.3,E2 -20347.3} C_VEL
LIN {X 0,Y 221.135,Z 351.685,A -85,B 0,C 180,E1 -20350.478,E2 -20350.478} C_VEL
LIN {X 0,Y 221.783,Z 353.955,A -85,B 0,C 180,E1 -20351.133,E2 -20351.133} C_VEL
LIN {X 0,Y 223.558,Z 356.196,A -85,B 0,C 180,E1 -20352.481,E2 -20352.481} C_VEL
LIN {X 0,Y 225.833,Z 357.588,A -85,B 0,C 180,E1 -20353.956,E2 -20353.956} C_VEL
LIN {X 0,Y 227.512,Z 360.661,A -85,B 0,C 180,E1 -20355.107,E2 -20355.107} C_VEL
LIN {X 0,Y 230.427,Z 363.375,A -85,B 0,C 180,E1 -20356.783,E2 -20356.783} C_VEL
LIN {X 0,Y 232.761,Z 366.836,A -85,B 0,C 180,E1 -20358.113,E2 -20358.113} C_VEL
LIN {X 0,Y 234.712,Z 368.751,A -85,B 0,C 180,E1 -20359.102,E2 -20359.102} C_VEL
LIN {X 0,Y 237.429,Z 372.435,A -85,B 0,C 180,E1 -20360.466,E2 -20360.466} C_VEL
LIN {X 0,Y 238.643,Z 373.942,A -85,B 0,C 180,E1 -20361.039,E2 -20361.039} C_VEL
LIN {X 0,Y 242.261,Z 378.759,A -85,B 0,C 180,E1 -20362.661,E2 -20362.661} C_VEL
LIN {X 0,Y 247.854,Z 386.449,A -85,B 0,C 180,E1 -20364.948,E2 -20364.948} C_VEL
LIN {X 0,Y 255.12,Z 397.538,A -85,B 0,C 180,E1 -20367.658,E2 -20367.658} C_VEL
LIN {X 0,Y 260.741,Z 408.09,A -85,B 0,C 180,E1 -20369.632,E2 -20369.632} C_VEL
LIN {X 0,Y 264.56,Z 416.031,A -85,B 0,C 180,E1 -20370.891,E2 -20370.891} C_VEL
LIN {X 0,Y 260.372,Z 482.964,A -85,B 0,C 180,E1 -20372.672,E2 -20372.672} C_VEL
LIN {X 0,Y 258.655,Z 497.446,A -85,B 0,C 180,E1 -20373.333,E2 -20373.333} C_VEL
LIN {X 0,Y 256.461,Z 510.381,A -85,B 0,C 180,E1 -20374.186,E2 -20374.186} C_VEL
LIN {X 0,Y 253.583,Z 523.727,A -85,B 0,C 180,E1 -20375.383,E2 -20375.383} C_VEL
LIN {X 0,Y 250.245,Z 536.213,A -85,B 0,C 180,E1 -20376.834,E2 -20376.834} C_VEL
LIN {X 0,Y 246.704,Z 547.227,A -85,B 0,C 180,E1 -20378.431,E2 -20378.431} C_VEL
LIN {X 0,Y 242.55,Z 558.544,A -85,B 0,C 180,E1 -20380.485,E2 -20380.485} C_VEL
LIN {X 0,Y 238.737,Z 567.904,A -85,B 0,C 180,E1 -20382.615,E2 -20382.615} C_VEL
LIN {X 0,Y 234.588,Z 577.211,A -85,B 0,C 180,E1 -20385.251,E2 -20385.251} C_VEL
LIN {X 0,Y 230.899,Z 584.813,A -85,B 0,C 180,E1 -20387.964,E2 -20387.964} C_VEL
LIN {X 0,Y 227.421,Z 591.59,A -85,B 0,C 180,E1 -20391.04,E2 -20391.04} C_VEL
LIN {X 0,Y 224.293,Z 597.417,A -85,B 0,C 180,E1 -20394.555,E2 -20394.555} C_VEL
LIN {X 0,Y 222.279,Z 601.048,A -85,B 0,C 180,E1 -20397.488,E2 -20397.488} C_VEL
LIN {X 0,Y 221.193,Z 602.9,A -85,B 0,C 180,E1 -20399.447,E2 -20399.447} C_VEL
LIN {X 0,Y 219.589,Z 605.385,A -85,B 0,C 180,E1 -20403.382,E2 -20403.382} C_VEL
LIN {X 0,Y 218.656,Z 606.365,A -85,B 0,C 180,E1 -20407.315,E2 -20407.315} C_VEL
LIN {X 0,Y 218.425,Z 606.305,A -85,B 0,C 180,E1 -20409.274,E2 -20409.274} C_VEL
LIN {X 0,Y 218.248,Z 605.112,A -85,B 0,C 180,E1 -20413.155,E2 -20413.155} C_VEL
LIN {X 0,Y 218.374,Z 603.977,A -85,B 0,C 180,E1 -20415.082,E2 -20415.082} C_VEL
LIN {X 0,Y 218.56,Z 602.483,A -85,B 0,C 180,E1 -20416.994,E2 -20416.994} C_VEL
LIN {X 0,Y 219.057,Z 599.502,A -85,B 0,C 180,E1 -20419.838,E2 -20419.838} C_VEL
LIN {X 0,Y 220.104,Z 594.215,A -85,B 0,C 180,E1 -20423.585,E2 -20423.585} C_VEL
LIN {X 0,Y 221.169,Z 589.094,A -85,B 0,C 180,E1 -20426.358,E2 -20426.358} C_VEL
LIN {X 0,Y 222.909,Z 581.768,A -85,B 0,C 180,E1 -20429.55,E2 -20429.55} C_VEL
LIN {X 0,Y 225.133,Z 572.828,A -85,B 0,C 180,E1 -20432.645,E2 -20432.645} C_VEL
LIN {X 0,Y 227.421,Z 563.18,A -85,B 0,C 180,E1 -20435.321,E2 -20435.321} C_VEL
LIN {X 0,Y 229.921,Z 552.617,A -85,B 0,C 180,E1 -20437.687,E2 -20437.687} C_VEL
LIN {X 0,Y 232.48,Z 540.944,A -85,B 0,C 180,E1 -20439.792,E2 -20439.792} C_VEL
LIN {X 0,Y 235.033,Z 527.97,A -85,B 0,C 180,E1 -20441.646,E2 -20441.646} C_VEL
LIN {X 0,Y 237.25,Z 514.307,A -85,B 0,C 180,E1 -20443.165,E2 -20443.165} C_VEL
LIN {X 0,Y 238.953,Z 501.147,A -85,B 0,C 180,E1 -20444.262,E2 -20444.262} C_VEL
LIN {X 0,Y 240.269,Z 486.854,A -85,B 0,C 180,E1 -20445.107,E2 -20445.107} C_VEL
LIN {X 0,Y 241.23,Z 471.078,A -85,B 0,C 180,E1 -20445.667,E2 -20445.667} C_VEL
LIN {X 0,Y 244.171,Z 399.408,A -85,B 0,C 180,E1 -20447.72,E2 -20447.72} C_VEL
LIN {X 0,Y 238.348,Z 384.488,A -85,B 0,C 180,E1 -20449.053,E2 -20449.053} C_VEL
LIN {X 0,Y 231.225,Z 370.595,A -85,B 0,C 180,E1 -20450.64,E2 -20450.64} C_VEL
LIN {X 0,Y 224.102,Z 358.071,A -85,B 0,C 180,E1 -20452.305,E2 -20452.305} C_VEL
LIN {X 0,Y 222.393,Z 355.168,A -85,B 0,C 180,E1 -20452.72,E2 -20452.72} C_VEL
LIN {X 0,Y 221.015,Z 352.484,A -85,B 0,C 180,E1 -20453.074,E2 -20453.074} C_VEL
LIN {X 0,Y 220.864,Z 351.603,A -85,B 0,C 180,E1 -20453.185,E2 -20453.185} C_VEL
LIN {X 0,Y 220.863,Z 351.599,A -85,B 0,C 180,E1 -20457.005,E2 -20457.005} C_VEL
LIN {X 0,Y 220.819,Z 351.606,A -85,B 0,C 180,E1 -20460.76,E2 -20460.76} C_VEL
LIN {X 0,Y 220.794,Z 351.6,A -85,B 0,C 180,E1 -20464.958,E2 -20464.958} C_VEL
LIN {X 0,Y 220.802,Z 351.591,A -85,B 0,C 180,E1 -20467.276,E2 -20467.276} C_VEL
LIN {X 0,Y 220.749,Z 351.607,A -85,B 0,C 180,E1 -20471.959,E2 -20471.959} C_VEL
LIN {X 0,Y 220.753,Z 351.592,A -85,B 0,C 180,E1 -20475.542,E2 -20475.542} C_VEL
LIN {X 0,Y 220.782,Z 351.602,A -85,B 0,C 180,E1 -20480.459,E2 -20480.459} C_VEL
LIN {X 0,Y 220.827,Z 351.575,A -85,B 0,C 180,E1 -20482.794,E2 -20482.794} C_VEL
LIN {X 0,Y 220.813,Z 351.598,A -85,B 0,C 180,E1 -20487.244,E2 -20487.244} C_VEL
LIN {X 0,Y 220.797,Z 351.601,A -85,B 0,C 180,E1 -20491.482,E2 -20491.482} C_VEL
LIN {X 0,Y 220.805,Z 351.604,A -85,B 0,C 180,E1 -20495.558,E2 -20495.558} C_VEL
LIN {X 0,Y 220.85,Z 351.594,A -85,B 0,C 180,E1 -20499.51,E2 -20499.51} C_VEL
LIN {X 0,Y 220.97,Z 351.58,A -85,B 0,C 180,E1 -20503.367,E2 -20503.367} C_VEL
LIN {X 0,Y 221.054,Z 351.546,A -85,B 0,C 180,E1 -20509.004,E2 -20509.004} C_VEL
LIN {X 0,Y 221.241,Z 351.549,A -85,B 0,C 180,E1 -20512.701,E2 -20512.701} C_VEL
LIN {X 0,Y 221.479,Z 351.493,A -85,B 0,C 180,E1 -20518.182,E2 -20518.182} C_VEL
LIN {X 0,Y 221.576,Z 351.475,A -85,B 0,C 180,E1 -20520.001,E2 -20520.001} C_VEL
LIN {X 0,Y 221.478,Z 351.501,A -85,B 0,C 180,E1 -20521.819,E2 -20521.819} C_VEL
LIN {X 0,Y 221.252,Z 351.547,A -85,B 0,C 180,E1 -20527.3,E2 -20527.3} C_VEL
LIN {X 0,Y 221.072,Z 351.571,A -85,B 0,C 180,E1 -20530.997,E2 -20530.997} C_VEL
LIN {X 0,Y 221.022,Z 351.578,A -85,B 0,C 180,E1 -20536.63,E2 -20536.63} C_VEL
LIN {X 0,Y 220.899,Z 351.588,A -85,B 0,C 180,E1 -20540.486,E2 -20540.486} C_VEL
LIN {X 0,Y 220.874,Z 351.589,A -85,B 0,C 180,E1 -20544.435,E2 -20544.435} C_VEL
LIN {X 0,Y 220.833,Z 351.598,A -85,B 0,C 180,E1 -20548.515,E2 -20548.515} C_VEL
LIN {X 0,Y 220.834,Z 351.597,A -85,B 0,C 180,E1 -20550.902,E2 -20550.902} C_VEL
LIN {X 0,Y 220.109,Z 351.69,A -85,B 0,C 180,E1 -20552.424,E2 -20552.424} C_VEL
LIN {X 0,Y 217.264,Z 352.046,A -85,B 0,C 180,E1 -20554.911,E2 -20554.911} C_VEL
LIN {X 0,Y 214.049,Z 352.434,A -85,B 0,C 180,E1 -20557.985,E2 -20557.985} C_VEL
LIN {X 0,Y 213.704,Z 352.476,A -85,B 0,C 180,E1 -20559.049,E2 -20559.049} C_VEL
LIN {X 0,Y 213.713,Z 352.488,A -85,B 0,C 180,E1 -20563.678,E2 -20563.678} C_VEL
LIN {X 0,Y 213.782,Z 352.623,A -85,B 0,C 180,E1 -20564.893,E2 -20564.893} C_VEL
LIN {X 0,Y 215.365,Z 358.477,A -85,B 0,C 180,E1 -20567.588,E2 -20567.588} C_VEL
LIN {X 0,Y 223.661,Z 375.517,A -85,B 0,C 180,E1 -20569.766,E2 -20569.766} C_VEL
LIN {X 0,Y 231.229,Z 393.592,A -85,B 0,C 180,E1 -20571.68,E2 -20571.68} C_VEL
LIN {X 0,Y 235.384,Z 405.067,A -85,B 0,C 180,E1 -20572.718,E2 -20572.718} C_VEL
LIN {X 0,Y 237.341,Z 422.468,A -85,B 0,C 180,E1 -20573.614,E2 -20573.614} C_VEL
LIN {X 0,Y 233.919,Z 497.665,A -85,B 0,C 180,E1 -20575.842,E2 -20575.842} C_VEL
LIN {X 0,Y 232.582,Z 512.241,A -85,B 0,C 180,E1 -20576.596,E2 -20576.596} C_VEL
LIN {X 0,Y 230.704,Z 526.229,A -85,B 0,C 180,E1 -20577.654,E2 -20577.654} C_VEL
LIN {X 0,Y 228.457,Z 539.258,A -85,B 0,C 180,E1 -20578.982,E2 -20578.982} C_VEL
LIN {X 0,Y 226.098,Z 551.167,A -85,B 0,C 180,E1 -20580.551,E2 -20580.551} C_VEL
LIN {X 0,Y 223.899,Z 561.107,A -85,B 0,C 180,E1 -20582.164,E2 -20582.164} C_VEL
LIN {X 0,Y 221.528,Z 571.127,A -85,B 0,C 180,E1 -20584.135,E2 -20584.135} C_VEL
LIN {X 0,Y 219.107,Z 580.488,A -85,B 0,C 180,E1 -20586.361,E2 -20586.361} C_VEL
LIN {X 0,Y 216.783,Z 589.864,A -85,B 0,C 180,E1 -20589.106,E2 -20589.106} C_VEL
LIN {X 0,Y 214.706,Z 598.418,A -85,B 0,C 180,E1 -20592.214,E2 -20592.214} C_VEL
LIN {X 0,Y 213.54,Z 604.128,A -85,B 0,C 180,E1 -20594.733,E2 -20594.733} C_VEL
LIN {X 0,Y 212.441,Z 609.414,A -85,B 0,C 180,E1 -20597.581,E2 -20597.581} C_VEL
LIN {X 0,Y 211.74,Z 614.979,A -85,B 0,C 180,E1 -20601.408,E2 -20601.408} C_VEL
LIN {X 0,Y 211.516,Z 619.045,A -85,B 0,C 180,E1 -20605.426,E2 -20605.426} C_VEL
LIN {X 0,Y 211.59,Z 620.858,A -85,B 0,C 180,E1 -20608.095,E2 -20608.095} C_VEL
LIN {X 0,Y 211.687,Z 621.735,A -85,B 0,C 180,E1 -20609.998,E2 -20609.998} C_VEL
LIN {X 0,Y 211.438,Z 622.441,A -85,B 0,C 180,E1 -20613.81,E2 -20613.81} C_VEL
LIN {X 0,Y 211.61,Z 621.824,A -85,B 0,C 180,E1 -20617.632,E2 -20617.632} C_VEL
LIN {X 0,Y 212.32,Z 619.899,A -85,B 0,C 180,E1 -20621.454,E2 -20621.454} C_VEL
LIN {X 0,Y 213.854,Z 616.635,A -85,B 0,C 180,E1 -20625.241,E2 -20625.241} C_VEL
LIN {X 0,Y 216.218,Z 611.92,A -85,B 0,C 180,E1 -20628.966,E2 -20628.966} C_VEL
LIN {X 0,Y 219.361,Z 605.624,A -85,B 0,C 180,E1 -20632.608,E2 -20632.608} C_VEL
LIN {X 0,Y 222.953,Z 598.664,A -85,B 0,C 180,E1 -20635.684,E2 -20635.684} C_VEL
LIN {X 0,Y 227.231,Z 590.085,A -85,B 0,C 180,E1 -20638.644,E2 -20638.644} C_VEL
LIN {X 0,Y 231.434,Z 581.162,A -85,B 0,C 180,E1 -20641.078,E2 -20641.078} C_VEL
LIN {X 0,Y 235.543,Z 571.563,A -85,B 0,C 180,E1 -20643.196,E2 -20643.196} C_VEL
LIN {X 0,Y 239.239,Z 561.883,A -85,B 0,C 180,E1 -20644.946,E2 -20644.946} C_VEL
LIN {X 0,Y 243.181,Z 550.527,A -85,B 0,C 180,E1 -20646.587,E2 -20646.587} C_VEL
LIN {X 0,Y 246.86,Z 538.137,A -85,B 0,C 180,E1 -20647.997,E2 -20647.997} C_VEL
LIN {X 0,Y 250.309,Z 524.312,A -85,B 0,C 180,E1 -20649.176,E2 -20649.176} C_VEL
LIN {X 0,Y 252.688,Z 511.947,A -85,B 0,C 180,E1 -20649.962,E2 -20649.962} C_VEL
LIN {X 0,Y 254.65,Z 497.213,A -85,B 0,C 180,E1 -20650.626,E2 -20650.626} C_VEL
LIN {X 0,Y 257.602,Z 452.891,A -85,B 0,C 180,E1 -20651.834,E2 -20651.834} C_VEL
LIN {X 0,Y 259.01,Z 428.152,A -85,B 0,C 180,E1 -20652.524,E2 -20652.524} C_VEL
LIN {X 0,Y 254.039,Z 416.551,A -85,B 0,C 180,E1 -20654.345,E2 -20654.345} C_VEL
LIN {X 0,Y 248.155,Z 404.657,A -85,B 0,C 180,E1 -20656.625,E2 -20656.625} C_VEL
LIN {X 0,Y 243.032,Z 395.474,A -85,B 0,C 180,E1 -20658.75,E2 -20658.75} C_VEL
LIN {X 0,Y 237.276,Z 385.961,A -85,B 0,C 180,E1 -20661.361,E2 -20661.361} C_VEL
LIN {X 0,Y 233.135,Z 379.628,A -85,B 0,C 180,E1 -20663.461,E2 -20663.461} C_VEL
LIN {X 0,Y 229.442,Z 374.121,A -85,B 0,C 180,E1 -20665.52,E2 -20665.52} C_VEL
LIN {X 0,Y 225.81,Z 369.073,A -85,B 0,C 180,E1 -20667.742,E2 -20667.742} C_VEL
LIN {X 0,Y 220.691,Z 362.342,A -85,B 0,C 180,E1 -20671.4,E2 -20671.4} C_VEL
LIN {X 0,Y 219.876,Z 361.146,A -85,B 0,C 180,E1 -20672.074,E2 -20672.074} C_VEL
LIN {X 0,Y 215.857,Z 356.638,A -85,B 0,C 180,E1 -20675.728,E2 -20675.728} C_VEL
LIN {X 0,Y 214.246,Z 354.138,A -85,B 0,C 180,E1 -20677.604,E2 -20677.604} C_VEL
LIN {X 0,Y 213.832,Z 352.464,A -85,B 0,C 180,E1 -20680.312,E2 -20680.312} C_VEL
LIN {X 0,Y 213.956,Z 352.459,A -85,B 0,C 180,E1 -20682.804,E2 -20682.804} C_VEL
LIN {X 0,Y 213.974,Z 352.456,A -85,B 0,C 180,E1 -20686.707,E2 -20686.707} C_VEL
LIN {X 0,Y 214.19,Z 352.426,A -85,B 0,C 180,E1 -20690.557,E2 -20690.557} C_VEL
LIN {X 0,Y 214.227,Z 352.413,A -85,B 0,C 180,E1 -20692.459,E2 -20692.459} C_VEL
LIN {X 0,Y 214.403,Z 352.393,A -85,B 0,C 180,E1 -20698.121,E2 -20698.121} C_VEL
LIN {X 0,Y 214.504,Z 352.384,A -85,B 0,C 180,E1 -20699.999,E2 -20699.999} C_VEL
LIN {X 0,Y 214.399,Z 352.392,A -85,B 0,C 180,E1 -20701.878,E2 -20701.878} C_VEL
LIN {X 0,Y 214.101,Z 352.573,A -85,B 0,C 180,E1 -20704.589,E2 -20704.589} C_VEL
LIN {X 0,Y 214.724,Z 354.652,A -85,B 0,C 180,E1 -20705.517,E2 -20705.517} C_VEL
LIN {X 0,Y 216.657,Z 357.001,A -85,B 0,C 180,E1 -20707.572,E2 -20707.572} C_VEL
LIN {X 0,Y 219.25,Z 358.574,A -85,B 0,C 180,E1 -20709.794,E2 -20709.794} C_VEL
LIN {X 0,Y 220.602,Z 361.422,A -85,B 0,C 180,E1 -20711.019,E2 -20711.019} C_VEL
LIN {X 0,Y 222.964,Z 363.647,A -85,B 0,C 180,E1 -20712.746,E2 -20712.746} C_VEL
LIN {X 0,Y 223.932,Z 364.372,A -85,B 0,C 180,E1 -20713.393,E2 -20713.393} C_VEL
LIN {X 0,Y 225.993,Z 367.607,A -85,B 0,C 180,E1 -20714.808,E2 -20714.808} C_VEL
LIN {X 0,Y 228.311,Z 369.834,A -85,B 0,C 180,E1 -20716.182,E2 -20716.182} C_VEL
LIN {X 0,Y 230.79,Z 373.373,A -85,B 0,C 180,E1 -20717.631,E2 -20717.631} C_VEL
LIN {X 0,Y 232.467,Z 375.151,A -85,B 0,C 180,E1 -20718.516,E2 -20718.516} C_VEL
LIN {X 0,Y 235.434,Z 379.039,A -85,B 0,C 180,E1 -20720.041,E2 -20720.041} C_VEL
LIN {X 0,Y 239.921,Z 385.272,A -85,B 0,C 180,E1 -20722.168,E2 -20722.168} C_VEL
LIN {X 0,Y 244.784,Z 392.053,A -85,B 0,C 180,E1 -20724.229,E2 -20724.229} C_VEL
LIN {X 0,Y 251.72,Z 402.838,A -85,B 0,C 180,E1 -20726.924,E2 -20726.924} C_VEL
LIN {X 0,Y 257.096,Z 413.246,A -85,B 0,C 180,E1 -20728.903,E2 -20728.903} C_VEL
LIN {X 0,Y 259.647,Z 418.815,A -85,B 0,C 180,E1 -20729.809,E2 -20729.809} C_VEL
LIN {X 0,Y 255.408,Z 483.689,A -85,B 0,C 180,E1 -20731.556,E2 -20731.556} C_VEL
LIN {X 0,Y 253.621,Z 498.025,A -85,B 0,C 180,E1 -20732.22,E2 -20732.22} C_VEL
LIN {X 0,Y 251.241,Z 511.502,A -85,B 0,C 180,E1 -20733.132,E2 -20733.132} C_VEL
LIN {X 0,Y 248.451,Z 523.792,A -85,B 0,C 180,E1 -20734.243,E2 -20734.243} C_VEL
LIN {X 0,Y 244.782,Z 537.008,A -85,B 0,C 180,E1 -20735.8,E2 -20735.8} C_VEL
LIN {X 0,Y 241.119,Z 547.925,A -85,B 0,C 180,E1 -20737.417,E2 -20737.417} C_VEL
LIN {X 0,Y 236.806,Z 559.174,A -85,B 0,C 180,E1 -20739.502,E2 -20739.502} C_VEL
LIN {X 0,Y 232.604,Z 568.961,A -85,B 0,C 180,E1 -20741.786,E2 -20741.786} C_VEL
LIN {X 0,Y 228.476,Z 577.725,A -85,B 0,C 180,E1 -20744.345,E2 -20744.345} C_VEL
LIN {X 0,Y 224.626,Z 585.286,A -85,B 0,C 180,E1 -20747.12,E2 -20747.12} C_VEL
LIN {X 0,Y 220.75,Z 592.354,A -85,B 0,C 180,E1 -20750.453,E2 -20750.453} C_VEL
LIN {X 0,Y 217.665,Z 597.736,A -85,B 0,C 180,E1 -20753.822,E2 -20753.822} C_VEL
LIN {X 0,Y 215.803,Z 600.859,A -85,B 0,C 180,E1 -20756.386,E2 -20756.386} C_VEL
LIN {X 0,Y 214.625,Z 602.816,A -85,B 0,C 180,E1 -20758.406,E2 -20758.406} C_VEL
LIN {X 0,Y 213.603,Z 604.361,A -85,B 0,C 180,E1 -20760.429,E2 -20760.429} C_VEL
LIN {X 0,Y 212.187,Z 606.236,A -85,B 0,C 180,E1 -20764.498,E2 -20764.498} C_VEL
LIN {X 0,Y 211.42,Z 606.621,A -85,B 0,C 180,E1 -20768.554,E2 -20768.554} C_VEL
LIN {X 0,Y 211.144,Z 605.566,A -85,B 0,C 180,E1 -20772.57,E2 -20772.57} C_VEL
LIN {X 0,Y 211.247,Z 604.389,A -85,B 0,C 180,E1 -20774.751,E2 -20774.751} C_VEL
LIN {X 0,Y 211.68,Z 601.296,A -85,B 0,C 180,E1 -20778.511,E2 -20778.511} C_VEL
LIN {X 0,Y 212.331,Z 597.869,A -85,B 0,C 180,E1 -20781.436,E2 -20781.436} C_VEL
LIN {X 0,Y 213.232,Z 593.566,A -85,B 0,C 180,E1 -20784.327,E2 -20784.327} C_VEL
LIN {X 0,Y 214.636,Z 587.276,A -85,B 0,C 180,E1 -20787.656,E2 -20787.656} C_VEL
LIN {X 0,Y 216.628,Z 579.42,A -85,B 0,C 180,E1 -20790.931,E2 -20790.931} C_VEL
LIN {X 0,Y 218.785,Z 571.211,A -85,B 0,C 180,E1 -20793.685,E2 -20793.685} C_VEL
LIN {X 0,Y 221.205,Z 561.344,A -85,B 0,C 180,E1 -20796.386,E2 -20796.386} C_VEL
LIN {X 0,Y 223.876,Z 550.354,A -85,B 0,C 180,E1 -20798.805,E2 -20798.805} C_VEL
LIN {X 0,Y 226.562,Z 538.158,A -85,B 0,C 180,E1 -20800.954,E2 -20800.954} C_VEL
LIN {X 0,Y 228.958,Z 526.063,A -85,B 0,C 180,E1 -20802.635,E2 -20802.635} C_VEL
LIN {X 0,Y 231.125,Z 512.712,A -85,B 0,C 180,E1 -20804.081,E2 -20804.081} C_VEL
LIN {X 0,Y 232.896,Z 498.427,A -85,B 0,C 180,E1 -20805.234,E2 -20805.234} C_VEL
LIN {X 0,Y 234.264,Z 483.535,A -85,B 0,C 180,E1 -20806.047,E2 -20806.047} C_VEL
LIN {X 0,Y 235.646,Z 455.511,A -85,B 0,C 180,E1 -20806.926,E2 -20806.926} C_VEL
LIN {X 0,Y 238.052,Z 401.668,A -85,B 0,C 180,E1 -20808.486,E2 -20808.486} C_VEL
LIN {X 0,Y 234.335,Z 391.604,A -85,B 0,C 180,E1 -20809.388,E2 -20809.388} C_VEL
LIN {X 0,Y 229.54,Z 381.138,A -85,B 0,C 180,E1 -20810.514,E2 -20810.514} C_VEL
LIN {X 0,Y 221.335,Z 366.131,A -85,B 0,C 180,E1 -20812.475,E2 -20812.475} C_VEL
LIN {X 0,Y 215.375,Z 356.096,A -85,B 0,C 180,E1 -20813.983,E2 -20813.983} C_VEL
LIN {X 0,Y 214.04,Z 353.601,A -85,B 0,C 180,E1 -20814.347,E2 -20814.347} C_VEL
LIN {X 0,Y 213.806,Z 352.481,A -85,B 0,C 180,E1 -20814.482,E2 -20814.482} C_VEL
LIN {X 0,Y 213.785,Z 352.481,A -85,B 0,C 180,E1 -20817.428,E2 -20817.428} C_VEL
LIN {X 0,Y 213.759,Z 352.481,A -85,B 0,C 180,E1 -20821.741,E2 -20821.741} C_VEL
LIN {X 0,Y 213.742,Z 352.468,A -85,B 0,C 180,E1 -20826.29,E2 -20826.29} C_VEL
LIN {X 0,Y 213.699,Z 352.489,A -85,B 0,C 180,E1 -20831.13,E2 -20831.13} C_VEL
LIN {X 0,Y 213.702,Z 352.466,A -85,B 0,C 180,E1 -20833.681,E2 -20833.681} C_VEL
LIN {X 0,Y 213.702,Z 352.476,A -85,B 0,C 180,E1 -20836.347,E2 -20836.347} C_VEL
LIN {X 0,Y 213.703,Z 352.478,A -85,B 0,C 180,E1 -20841.33,E2 -20841.33} C_VEL
LIN {X 0,Y 213.755,Z 352.466,A -85,B 0,C 180,E1 -20846.018,E2 -20846.018} C_VEL
LIN {X 0,Y 213.749,Z 352.483,A -85,B 0,C 180,E1 -20850.45,E2 -20850.45} C_VEL
LIN {X 0,Y 213.753,Z 352.485,A -85,B 0,C 180,E1 -20854.696,E2 -20854.696} C_VEL
LIN {X 0,Y 213.778,Z 352.473,A -85,B 0,C 180,E1 -20858.801,E2 -20858.801} C_VEL
LIN {X 0,Y 213.882,Z 352.463,A -85,B 0,C 180,E1 -20862.799,E2 -20862.799} C_VEL
LIN {X 0,Y 213.916,Z 352.426,A -85,B 0,C 180,E1 -20866.705,E2 -20866.705} C_VEL
LIN {X 0,Y 214.132,Z 352.421,A -85,B 0,C 180,E1 -20870.555,E2 -20870.555} C_VEL
LIN {X 0,Y 214.084,Z 352.44,A -85,B 0,C 180,E1 -20874.349,E2 -20874.349} C_VEL
LIN {X 0,Y 214.416,Z 352.372,A -85,B 0,C 180,E1 -20878.122,E2 -20878.122} C_VEL
LIN {X 0,Y 214.541,Z 352.349,A -85,B 0,C 180,E1 -20880.001,E2 -20880.001} C_VEL
LIN {X 0,Y 214.415,Z 352.38,A -85,B 0,C 180,E1 -20881.879,E2 -20881.879} C_VEL
LIN {X 0,Y 214.193,Z 352.424,A -85,B 0,C 180,E1 -20887.542,E2 -20887.542} C_VEL
LIN {X 0,Y 214.004,Z 352.453,A -85,B 0,C 180,E1 -20891.365,E2 -20891.365} C_VEL
LIN {X 0,Y 213.938,Z 352.457,A -85,B 0,C 180,E1 -20895.237,E2 -20895.237} C_VEL
LIN {X 0,Y 213.846,Z 352.463,A -85,B 0,C 180,E1 -20899.187,E2 -20899.187} C_VEL
LIN {X 0,Y 213.854,Z 352.47,A -85,B 0,C 180,E1 -20903.227,E2 -20903.227} C_VEL
LIN {X 0,Y 213.835,Z 352.473,A -85,B 0,C 180,E1 -20907.45,E2 -20907.45} C_VEL
LIN {X 0,Y 213.773,Z 352.481,A -85,B 0,C 180,E1 -20911.737,E2 -20911.737} C_VEL
LIN {X 0,Y 213.749,Z 352.482,A -85,B 0,C 180,E1 -20916.288,E2 -20916.288} C_VEL
LIN {X 0,Y 213.704,Z 352.476,A -85,B 0,C 180,E1 -20919.049,E2 -20919.049} C_VEL
LIN {X 0,Y 212.935,Z 352.588,A -85,B 0,C 180,E1 -20920.132,E2 -20920.132} C_VEL
LIN {X 0,Y 207.315,Z 353.595,A -85,B 0,C 180,E1 -20923.521,E2 -20923.521} C_VEL
LIN {X 0,Y 207.031,Z 354.734,A -85,B 0,C 180,E1 -20924.447,E2 -20924.447} C_VEL
LIN {X 0,Y 207.075,Z 354.883,A -85,B 0,C 180,E1 -20924.525,E2 -20924.525} C_VEL
LIN {X 0,Y 208.078,Z 358.406,A -85,B 0,C 180,E1 -20926.13,E2 -20926.13} C_VEL
LIN {X 0,Y 215.097,Z 372.257,A -85,B 0,C 180,E1 -20928.104,E2 -20928.104} C_VEL
LIN {X 0,Y 222.281,Z 388.241,A -85,B 0,C 180,E1 -20930.028,E2 -20930.028} C_VEL
LIN {X 0,Y 229.337,Z 406.846,A -85,B 0,C 180,E1 -20931.88,E2 -20931.88} C_VEL
LIN {X 0,Y 231.196,Z 422.843,A -85,B 0,C 180,E1 -20932.749,E2 -20932.749} C_VEL
LIN {X 0,Y 227.738,Z 496.79,A -85,B 0,C 180,E1 -20934.983,E2 -20934.983} C_VEL
LIN {X 0,Y 226.449,Z 510.815,A -85,B 0,C 180,E1 -20935.701,E2 -20935.701} C_VEL
LIN {X 0,Y 224.483,Z 525.092,A -85,B 0,C 180,E1 -20936.777,E2 -20936.777} C_VEL
LIN {X 0,Y 222.312,Z 537.412,A -85,B 0,C 180,E1 -20938.025,E2 -20938.025} C_VEL
LIN {X 0,Y 219.71,Z 550.309,A -85,B 0,C 180,E1 -20939.732,E2 -20939.732} C_VEL
LIN {X 0,Y 217.29,Z 560.986,A -85,B 0,C 180,E1 -20941.504,E2 -20941.504} C_VEL
LIN {X 0,Y 214.562,Z 571.972,A -85,B 0,C 180,E1 -20943.754,E2 -20943.754} C_VEL
LIN {X 0,Y 212.103,Z 581.152,A -85,B 0,C 180,E1 -20946.051,E2 -20946.051} C_VEL
LIN {X 0,Y 209.723,Z 590.372,A -85,B 0,C 180,E1 -20948.883,E2 -20948.883} C_VEL
LIN {X 0,Y 207.783,Z 597.976,A -85,B 0,C 180,E1 -20951.745,E2 -20951.745} C_VEL
LIN {X 0,Y 206.22,Z 605.32,A -85,B 0,C 180,E1 -20955.189,E2 -20955.189} C_VEL
LIN {X 0,Y 205.196,Z 610.38,A -85,B 0,C 180,E1 -20958.139,E2 -20958.139} C_VEL
LIN {X 0,Y 204.592,Z 615.576,A -85,B 0,C 180,E1 -20962.101,E2 -20962.101} C_VEL
LIN {X 0,Y 204.415,Z 618.868,A -85,B 0,C 180,E1 -20965.604,E2 -20965.604} C_VEL
LIN {X 0,Y 204.504,Z 620.468,A -85,B 0,C 180,E1 -20968.029,E2 -20968.029} C_VEL
LIN {X 0,Y 204.598,Z 621.38,A -85,B 0,C 180,E1 -20969.998,E2 -20969.998} C_VEL
LIN {X 0,Y 204.462,Z 621.935,A -85,B 0,C 180,E1 -20971.968,E2 -20971.968} C_VEL
LIN {X 0,Y 204.39,Z 622.043,A -85,B 0,C 180,E1 -20975.919,E2 -20975.919} C_VEL
LIN {X 0,Y 204.855,Z 620.842,A -85,B 0,C 180,E1 -20979.875,E2 -20979.875} C_VEL
LIN {X 0,Y 205.987,Z 618.326,A -85,B 0,C 180,E1 -20983.816,E2 -20983.816} C_VEL
LIN {X 0,Y 208.114,Z 614.444,A -85,B 0,C 180,E1 -20987.692,E2 -20987.692} C_VEL
LIN {X 0,Y 211.012,Z 609.059,A -85,B 0,C 180,E1 -20991.49,E2 -20991.49} C_VEL
LIN {X 0,Y 213.804,Z 603.933,A -85,B 0,C 180,E1 -20994.259,E2 -20994.259} C_VEL
LIN {X 0,Y 217.798,Z 596.646,A -85,B 0,C 180,E1 -20997.374,E2 -20997.374} C_VEL
LIN {X 0,Y 222.434,Z 587.677,A -85,B 0,C 180,E1 -21000.365,E2 -21000.365} C_VEL
LIN {X 0,Y 226.934,Z 578.314,A -85,B 0,C 180,E1 -21002.815,E2 -21002.815} C_VEL
LIN {X 0,Y 231.108,Z 568.584,A -85,B 0,C 180,E1 -21004.882,E2 -21004.882} C_VEL
LIN {X 0,Y 235.713,Z 556.685,A -85,B 0,C 180,E1 -21006.871,E2 -21006.871} C_VEL
LIN {X 0,Y 239.863,Z 544.209,A -85,B 0,C 180,E1 -21008.506,E2 -21008.506} C_VEL
LIN {X 0,Y 243.382,Z 532.132,A -85,B 0,C 180,E1 -21009.707,E2 -21009.707} C_VEL
LIN {X 0,Y 246.64,Z 517.659,A -85,B 0,C 180,E1 -21010.811,E2 -21010.811} C_VEL
LIN {X 0,Y 249.072,Z 503.732,A -85,B 0,C 180,E1 -21011.534,E2 -21011.534} C_VEL
LIN {X 0,Y 250.523,Z 489.507,A -85,B 0,C 180,E1 -21012.047,E2 -21012.047} C_VEL
LIN {X 0,Y 254.251,Z 430.772,A -85,B 0,C 180,E1 -21013.65,E2 -21013.65} C_VEL
LIN {X 0,Y 250.009,Z 420.67,A -85,B 0,C 180,E1 -21015.303,E2 -21015.303} C_VEL
LIN {X 0,Y 244.729,Z 409.777,A -85,B 0,C 180,E1 -21017.452,E2 -21017.452} C_VEL
LIN {X 0,Y 239.722,Z 400.609,A -85,B 0,C 180,E1 -21019.63,E2 -21019.63} C_VEL
LIN {X 0,Y 235.955,Z 394.239,A -85,B 0,C 180,E1 -21021.401,E2 -21021.401} C_VEL
LIN {X 0,Y 231.051,Z 386.153,A -85,B 0,C 180,E1 -21023.971,E2 -21023.971} C_VEL
LIN {X 0,Y 227.097,Z 380.23,A -85,B 0,C 180,E1 -21026.256,E2 -21026.256} C_VEL
LIN {X 0,Y 222.875,Z 374.247,A -85,B 0,C 180,E1 -21028.993,E2 -21028.993} C_VEL
LIN {X 0,Y 218.901,Z 368.787,A -85,B 0,C 180,E1 -21032.033,E2 -21032.033} C_VEL
LIN {X 0,Y 218.038,Z 367.58,A -85,B 0,C 180,E1 -21032.774,E2 -21032.774} C_VEL
LIN {X 0,Y 214.296,Z 363.199,A -85,B 0,C 180,E1 -21036.38,E2 -21036.38} C_VEL
LIN {X 0,Y 212.459,Z 360.407,A -85,B 0,C 180,E1 -21038.661,E2 -21038.661} C_VEL
LIN {X 0,Y 211.11,Z 359.001,A -85,B 0,C 180,E1 -21040.554,E2 -21040.554} C_VEL
LIN {X 0,Y 207.717,Z 355.313,A -85,B 0,C 180,E1 -21050.26,E2 -21050.26} C_VEL
LIN {X 0,Y 207.745,Z 355.365,A -85,B 0,C 180,E1 -21052.711,E2 -21052.711} C_VEL
LIN {X 0,Y 210.205,Z 358.076,A -85,B 0,C 180,E1 -21060.526,E2 -21060.526} C_VEL
LIN {X 0,Y 212.676,Z 359.576,A -85,B 0,C 180,E1 -21064.026,E2 -21064.026} C_VEL
LIN {X 0,Y 213.779,Z 362.089,A -85,B 0,C 180,E1 -21065.541,E2 -21065.541} C_VEL
LIN {X 0,Y 216.372,Z 364.604,A -85,B 0,C 180,E1 -21068.169,E2 -21068.169} C_VEL
LIN {X 0,Y 217.602,Z 365.417,A -85,B 0,C 180,E1 -21069.234,E2 -21069.234} C_VEL
LIN {X 0,Y 219.28,Z 368.472,A -85,B 0,C 180,E1 -21070.766,E2 -21070.766} C_VEL
LIN {X 0,Y 222.108,Z 371.08,A -85,B 0,C 180,E1 -21072.848,E2 -21072.848} C_VEL
LIN {X 0,Y 224.59,Z 374.655,A -85,B 0,C 180,E1 -21074.573,E2 -21074.573} C_VEL
LIN {X 0,Y 226.284,Z 376.386,A -85,B 0,C 180,E1 -21075.611,E2 -21075.611} C_VEL
LIN {X 0,Y 229.083,Z 380.153,A -85,B 0,C 180,E1 -21077.276,E2 -21077.276} C_VEL
LIN {X 0,Y 230.419,Z 381.819,A -85,B 0,C 180,E1 -21078.016,E2 -21078.016} C_VEL
LIN {X 0,Y 234.44,Z 387.321,A -85,B 0,C 180,E1 -21080.13,E2 -21080.13} C_VEL
LIN {X 0,Y 237.707,Z 391.899,A -85,B 0,C 180,E1 -21081.712,E2 -21081.712} C_VEL
LIN {X 0,Y 242.052,Z 398.175,A -85,B 0,C 180,E1 -21083.622,E2 -21083.622} C_VEL
LIN {X 0,Y 248.323,Z 408.101,A -85,B 0,C 180,E1 -21086.157,E2 -21086.157} C_VEL
LIN {X 0,Y 253.604,Z 418.59,A -85,B 0,C 180,E1 -21088.188,E2 -21088.188} C_VEL
LIN {X 0,Y 254.803,Z 421.2,A -85,B 0,C 180,E1 -21088.636,E2 -21088.636} C_VEL
LIN {X 0,Y 250.689,Z 483.39,A -85,B 0,C 180,E1 -21090.352,E2 -21090.352} C_VEL
LIN {X 0,Y 248.808,Z 498.01,A -85,B 0,C 180,E1 -21091.024,E2 -21091.024} C_VEL
LIN {X 0,Y 246.36,Z 511.439,A -85,B 0,C 180,E1 -21091.934,E2 -21091.934} C_VEL
LIN {X 0,Y 243.321,Z 524.341,A -85,B 0,C 180,E1 -21093.113,E2 -21093.113} C_VEL
LIN {X 0,Y 239.829,Z 536.459,A -85,B 0,C 180,E1 -21094.542,E2 -21094.542} C_VEL
LIN {X 0,Y 235.619,Z 548.631,A -85,B 0,C 180,E1 -21096.359,E2 -21096.359} C_VEL
LIN {X 0,Y 231.133,Z 559.804,A -85,B 0,C 180,E1 -21098.47,E2 -21098.47} C_VEL
LIN {X 0,Y 226.912,Z 569.188,A -85,B 0,C 180,E1 -21100.701,E2 -21100.701} C_VEL
LIN {X 0,Y 222.431,Z 578.238,A -85,B 0,C 180,E1 -21103.391,E2 -21103.391} C_VEL
LIN {X 0,Y 218.38,Z 585.753,A -85,B 0,C 180,E1 -21106.22,E2 -21106.22} C_VEL
LIN {X 0,Y 214.836,Z 591.873,A -85,B 0,C 180,E1 -21109.139,E2 -21109.139} C_VEL
LIN {X 0,Y 211.88,Z 596.803,A -85,B 0,C 180,E1 -21112.151,E2 -21112.151} C_VEL
LIN {X 0,Y 209.437,Z 600.669,A -85,B 0,C 180,E1 -21115.22,E2 -21115.22} C_VEL
LIN {X 0,Y 207.859,Z 603.067,A -85,B 0,C 180,E1 -21117.701,E2 -21117.701} C_VEL
LIN {X 0,Y 206.038,Z 605.558,A -85,B 0,C 180,E1 -21121.477,E2 -21121.477} C_VEL
LIN {X 0,Y 204.798,Z 606.859,A -85,B 0,C 180,E1 -21125.684,E2 -21125.684} C_VEL
LIN {X 0,Y 204.172,Z 606.657,A -85,B 0,C 180,E1 -21129.868,E2 -21129.868} C_VEL
LIN {X 0,Y 204.099,Z 605.02,A -85,B 0,C 180,E1 -21134.012,E2 -21134.012} C_VEL
LIN {X 0,Y 204.495,Z 601.95,A -85,B 0,C 180,E1 -21138.102,E2 -21138.102} C_VEL
LIN {X 0,Y 205.157,Z 598.662,A -85,B 0,C 180,E1 -21141.134,E2 -21141.134} C_VEL
LIN {X 0,Y 206.047,Z 594.504,A -85,B 0,C 180,E1 -21144.129,E2 -21144.129} C_VEL
LIN {X 0,Y 207.233,Z 589.32,A -85,B 0,C 180,E1 -21147.086,E2 -21147.086} C_VEL
LIN {X 0,Y 209.141,Z 581.919,A -85,B 0,C 180,E1 -21150.483,E2 -21150.483} C_VEL
LIN {X 0,Y 211.635,Z 572.712,A -85,B 0,C 180,E1 -21153.81,E2 -21153.81} C_VEL
LIN {X 0,Y 214.11,Z 563.083,A -85,B 0,C 180,E1 -21156.599,E2 -21156.599} C_VEL
LIN {X 0,Y 216.805,Z 552.393,A -85,B 0,C 180,E1 -21159.094,E2 -21159.094} C_VEL
LIN {X 0,Y 219.577,Z 540.557,A -85,B 0,C 180,E1 -21161.307,E2 -21161.307} C_VEL
LIN {X 0,Y 222.023,Z 528.957,A -85,B 0,C 180,E1 -21163.036,E2 -21163.036} C_VEL
LIN {X 0,Y 224.263,Z 516.379,A -85,B 0,C 180,E1 -21164.521,E2 -21164.521} C_VEL
LIN {X 0,Y 226.2,Z 502.433,A -85,B 0,C 180,E1 -21165.777,E2 -21165.777} C_VEL
LIN {X 0,Y 227.645,Z 488.462,A -85,B 0,C 180,E1 -21166.665,E2 -21166.665} C_VEL
LIN {X 0,Y 228.661,Z 473.305,A -85,B 0,C 180,E1 -21167.252,E2 -21167.252} C_VEL
LIN {X 0,Y 231.792,Z 402.765,A -85,B 0,C 180,E1 -21169.362,E2 -21169.362} C_VEL
LIN {X 0,Y 226.542,Z 389.679,A -85,B 0,C 180,E1 -21170.674,E2 -21170.674} C_VEL
LIN {X 0,Y 218.202,Z 373.602,A -85,B 0,C 180,E1 -21172.739,E2 -21172.739} C_VEL
LIN {X 0,Y 210.837,Z 360.935,A -85,B 0,C 180,E1 -21174.668,E2 -21174.668} C_VEL
LIN {X 0,Y 208.48,Z 357.205,A -85,B 0,C 180,E1 -21175.306,E2 -21175.306} C_VEL
LIN {X 0,Y 206.951,Z 354.46,A -85,B 0,C 180,E1 -21175.744,E2 -21175.744} C_VEL
LIN {X 0,Y 206.722,Z 353.361,A -85,B 0,C 180,E1 -21175.869,E2 -21175.869} C_VEL
LIN {X 0,Y 206.696,Z 353.365,A -85,B 0,C 180,E1 -21180.667,E2 -21180.667} C_VEL
LIN {X 0,Y 206.7,Z 353.351,A -85,B 0,C 180,E1 -21185.313,E2 -21185.313} C_VEL
LIN {X 0,Y 206.648,Z 353.37,A -85,B 0,C 180,E1 -21190.256,E2 -21190.256} C_VEL
LIN {X 0,Y 206.631,Z 353.343,A -85,B 0,C 180,E1 -21194.419,E2 -21194.419} C_VEL
LIN {X 0,Y 206.631,Z 353.369,A -85,B 0,C 180,E1 -21198.443,E2 -21198.443} C_VEL
LIN {X 0,Y 206.665,Z 353.341,A -85,B 0,C 180,E1 -21202.258,E2 -21202.258} C_VEL
LIN {X 0,Y 206.702,Z 353.328,A -85,B 0,C 180,E1 -21204.69,E2 -21204.69} C_VEL
LIN {X 0,Y 206.697,Z 353.362,A -85,B 0,C 180,E1 -21209.336,E2 -21209.336} C_VEL
LIN {X 0,Y 206.688,Z 353.359,A -85,B 0,C 180,E1 -21213.767,E2 -21213.767} C_VEL
LIN {X 0,Y 206.716,Z 353.352,A -85,B 0,C 180,E1 -21218.039,E2 -21218.039} C_VEL
LIN {X 0,Y 206.807,Z 353.348,A -85,B 0,C 180,E1 -21222.191,E2 -21222.191} C_VEL
LIN {X 0,Y 206.856,Z 353.307,A -85,B 0,C 180,E1 -21226.242,E2 -21226.242} C_VEL
LIN {X 0,Y 207.078,Z 353.296,A -85,B 0,C 180,E1 -21230.231,E2 -21230.231} C_VEL
LIN {X 0,Y 207.047,Z 353.318,A -85,B 0,C 180,E1 -21234.156,E2 -21234.156} C_VEL
LIN {X 0,Y 207.356,Z 353.25,A -85,B 0,C 180,E1 -21238.058,E2 -21238.058} C_VEL
LIN {X 0,Y 207.507,Z 353.223,A -85,B 0,C 180,E1 -21240.001,E2 -21240.001} C_VEL
LIN {X 0,Y 207.057,Z 353.312,A -85,B 0,C 180,E1 -21243.893,E2 -21243.893} C_VEL
LIN {X 0,Y 207.137,Z 353.301,A -85,B 0,C 180,E1 -21247.801,E2 -21247.801} C_VEL
LIN {X 0,Y 206.929,Z 353.334,A -85,B 0,C 180,E1 -21251.759,E2 -21251.759} C_VEL
LIN {X 0,Y 206.872,Z 353.34,A -85,B 0,C 180,E1 -21255.771,E2 -21255.771} C_VEL
LIN {X 0,Y 206.79,Z 353.341,A -85,B 0,C 180,E1 -21259.869,E2 -21259.869} C_VEL
LIN {X 0,Y 206.77,Z 353.346,A -85,B 0,C 180,E1 -21264.072,E2 -21264.072} C_VEL
LIN {X 0,Y 206.743,Z 353.353,A -85,B 0,C 180,E1 -21268.42,E2 -21268.42} C_VEL
LIN {X 0,Y 206.704,Z 353.358,A -85,B 0,C 180,E1 -21272.957,E2 -21272.957} C_VEL
LIN {X 0,Y 206.684,Z 353.349,A -85,B 0,C 180,E1 -21277.74,E2 -21277.74} C_VEL
LIN {X 0,Y 206.648,Z 353.368,A -85,B 0,C 180,E1 -21281.562,E2 -21281.562} C_VEL
LIN {X 0,Y 206.72,Z 353.556,A -85,B 0,C 180,E1 -21283.869,E2 -21283.869} C_VEL
LIN {X 0,Y 207.075,Z 354.883,A -85,B 0,C 180,E1 -21284.525,E2 -21284.525} C_VEL
LIN {X 0,Y 207.709,Z 357.23,A -85,B 0,C 180,E1 -21285.347,E2 -21285.347} C_VEL
LIN {X 0,Y 208.647,Z 362.018,A -85,B 0,C 180,E1 -21286.232,E2 -21286.232} C_VEL
LIN {X 0,Y 209.511,Z 367.513,A -85,B 0,C 180,E1 -21286.817,E2 -21286.817} C_VEL
LIN {X 0,Y 210.851,Z 375.461,A -85,B 0,C 180,E1 -21287.421,E2 -21287.421} C_VEL
LIN {X 0,Y 212.391,Z 381.143,A -85,B 0,C 180,E1 -21287.957,E2 -21287.957} C_VEL
LIN {X 0,Y 213.138,Z 382.897,A -85,B 0,C 180,E1 -21288.172,E2 -21288.172} C_VEL
LIN {X 0,Y 220.162,Z 400.03,A -85,B 0,C 180,E1 -21290.13,E2 -21290.13} C_VEL
LIN {X 0,Y 223.596,Z 409.8,A -85,B 0,C 180,E1 -21291.084,E2 -21291.084} C_VEL
LIN {X 0,Y 225.093,Z 423.42,A -85,B 0,C 180,E1 -21291.843,E2 -21291.843} C_VEL
LIN {X 0,Y 221.493,Z 497.09,A -85,B 0,C 180,E1 -21294.123,E2 -21294.123} C_VEL
LIN {X 0,Y 220.048,Z 511.672,A -85,B 0,C 180,E1 -21294.906,E2 -21294.906} C_VEL
LIN {X 0,Y 217.973,Z 526.248,A -85,B 0,C 180,E1 -21296.067,E2 -21296.067} C_VEL
LIN {X 0,Y 215.586,Z 539.16,A -85,B 0,C 180,E1 -21297.458,E2 -21297.458} C_VEL
LIN {X 0,Y 213.014,Z 551.072,A -85,B 0,C 180,E1 -21299.114,E2 -21299.114} C_VEL
LIN {X 0,Y 210.711,Z 560.865,A -85,B 0,C 180,E1 -21300.802,E2 -21300.802} C_VEL
LIN {X 0,Y 208.136,Z 570.832,A -85,B 0,C 180,E1 -21302.879,E2 -21302.879} C_VEL
LIN {X 0,Y 205.553,Z 580.155,A -85,B 0,C 180,E1 -21305.237,E2 -21305.237} C_VEL
LIN {X 0,Y 203.04,Z 589.498,A -85,B 0,C 180,E1 -21308.153,E2 -21308.153} C_VEL
LIN {X 0,Y 201.097,Z 596.661,A -85,B 0,C 180,E1 -21310.866,E2 -21310.866} C_VEL
LIN {X 0,Y 199.689,Z 602.695,A -85,B 0,C 180,E1 -21313.645,E2 -21313.645} C_VEL
LIN {X 0,Y 198.477,Z 608.165,A -85,B 0,C 180,E1 -21316.692,E2 -21316.692} C_VEL
LIN {X 0,Y 197.636,Z 613.9,A -85,B 0,C 180,E1 -21320.79,E2 -21320.79} C_VEL
LIN {X 0,Y 197.388,Z 617.11,A -85,B 0,C 180,E1 -21323.866,E2 -21323.866} C_VEL
LIN {X 0,Y 197.402,Z 620.075,A -85,B 0,C 180,E1 -21327.958,E2 -21327.958} C_VEL
LIN {X 0,Y 197.512,Z 621.023,A -85,B 0,C 180,E1 -21329.998,E2 -21329.998} C_VEL
LIN {X 0,Y 197.253,Z 621.865,A -85,B 0,C 180,E1 -21334.084,E2 -21334.084} C_VEL
LIN {X 0,Y 197.482,Z 621.387,A -85,B 0,C 180,E1 -21338.182,E2 -21338.182} C_VEL
LIN {X 0,Y 198.342,Z 619.602,A -85,B 0,C 180,E1 -21342.273,E2 -21342.273} C_VEL
LIN {X 0,Y 200.125,Z 616.486,A -85,B 0,C 180,E1 -21346.315,E2 -21346.315} C_VEL
LIN {X 0,Y 202.702,Z 611.958,A -85,B 0,C 180,E1 -21350.284,E2 -21350.284} C_VEL
LIN {X 0,Y 206.282,Z 605.868,A -85,B 0,C 180,E1 -21354.13,E2 -21354.13} C_VEL
LIN {X 0,Y 210.21,Z 599.092,A -85,B 0,C 180,E1 -21357.366,E2 -21357.366} C_VEL
LIN {X 0,Y 214.897,Z 590.717,A -85,B 0,C 180,E1 -21360.456,E2 -21360.456} C_VEL
LIN {X 0,Y 219.441,Z 582.028,A -85,B 0,C 180,E1 -21362.985,E2 -21362.985} C_VEL
LIN {X 0,Y 224.191,Z 571.905,A -85,B 0,C 180,E1 -21365.343,E2 -21365.343} C_VEL
LIN {X 0,Y 228.297,Z 562.225,A -85,B 0,C 180,E1 -21367.165,E2 -21367.165} C_VEL
LIN {X 0,Y 232.522,Z 551.089,A -85,B 0,C 180,E1 -21368.839,E2 -21368.839} C_VEL
LIN {X 0,Y 236.469,Z 538.99,A -85,B 0,C 180,E1 -21370.27,E2 -21370.27} C_VEL
LIN {X 0,Y 240.142,Z 525.583,A -85,B 0,C 180,E1 -21371.461,E2 -21371.461} C_VEL
LIN {X 0,Y 242.64,Z 513.89,A -85,B 0,C 180,E1 -21372.26,E2 -21372.26} C_VEL
LIN {X 0,Y 244.912,Z 499.272,A -85,B 0,C 180,E1 -21372.961,E2 -21372.961} C_VEL
LIN {X 0,Y 246.533,Z 479.747,A -85,B 0,C 180,E1 -21373.559,E2 -21373.559} C_VEL
LIN {X 0,Y 249.634,Z 433.455,A -85,B 0,C 180,E1 -21374.815,E2 -21374.815} C_VEL
LIN {X 0,Y 245.129,Z 422.734,A -85,B 0,C 180,E1 -21376.679,E2 -21376.679} C_VEL
LIN {X 0,Y 240.279,Z 412.741,A -85,B 0,C 180,E1 -21378.784,E2 -21378.784} C_VEL
LIN {X 0,Y 236.139,Z 405.133,A -85,B 0,C 180,E1 -21380.695,E2 -21380.695} C_VEL
LIN {X 0,Y 231.239,Z 396.585,A -85,B 0,C 180,E1 -21383.222,E2 -21383.222} C_VEL
LIN {X 0,Y 227.826,Z 391.017,A -85,B 0,C 180,E1 -21385.15,E2 -21385.15} C_VEL
LIN {X 0,Y 224.844,Z 386.342,A -85,B 0,C 180,E1 -21386.978,E2 -21386.978} C_VEL
LIN {X 0,Y 220.911,Z 380.59,A -85,B 0,C 180,E1 -21389.649,E2 -21389.649} C_VEL
LIN {X 0,Y 217.112,Z 375.156,A -85,B 0,C 180,E1 -21392.715,E2 -21392.715} C_VEL
LIN {X 0,Y 216.12,Z 373.918,A -85,B 0,C 180,E1 -21393.602,E2 -21393.602} C_VEL
LIN {X 0,Y 213.081,Z 370.106,A -85,B 0,C 180,E1 -21396.684,E2 -21396.684} C_VEL
LIN {X 0,Y 211.239,Z 367.259,A -85,B 0,C 180,E1 -21399.043,E2 -21399.043} C_VEL
LIN {X 0,Y 209.929,Z 365.925,A -85,B 0,C 180,E1 -21400.948,E2 -21400.948} C_VEL
LIN {X 0,Y 206.829,Z 362.38,A -85,B 0,C 180,E1 -21410.217,E2 -21410.217} C_VEL
LIN {X 0,Y 206.849,Z 362.431,A -85,B 0,C 180,E1 -21412.679,E2 -21412.679} C_VEL
LIN {X 0,Y 209.557,Z 365.327,A -85,B 0,C 180,E1 -21420.96,E2 -21420.96} C_VEL
LIN {X 0,Y 211.359,Z 366.554,A -85,B 0,C 180,E1 -21423.555,E2 -21423.555} C_VEL
LIN {X 0,Y 212.862,Z 369.467,A -85,B 0,C 180,E1 -21425.58,E2 -21425.58} C_VEL
LIN {X 0,Y 215.804,Z 371.872,A -85,B 0,C 180,E1 -21428.485,E2 -21428.485} C_VEL
LIN {X 0,Y 217.983,Z 375.475,A -85,B 0,C 180,E1 -21430.508,E2 -21430.508} C_VEL
LIN {X 0,Y 220.343,Z 377.774,A -85,B 0,C 180,E1 -21432.316,E2 -21432.316} C_VEL
LIN {X 0,Y 223.032,Z 381.443,A -85,B 0,C 180,E1 -21434.226,E2 -21434.226} C_VEL
LIN {X 0,Y 224.382,Z 383.025,A -85,B 0,C 180,E1 -21435.091,E2 -21435.091} C_VEL
LIN {X 0,Y 227.398,Z 386.941,A -85,B 0,C 180,E1 -21436.924,E2 -21436.924} C_VEL
LIN {X 0,Y 232.049,Z 393.496,A -85,B 0,C 180,E1 -21439.497,E2 -21439.497} C_VEL
LIN {X 0,Y 236.891,Z 400.448,A -85,B 0,C 180,E1 -21441.889,E2 -21441.889} C_VEL
LIN {X 0,Y 243.466,Z 410.827,A -85,B 0,C 180,E1 -21444.754,E2 -21444.754} C_VEL
LIN {X 0,Y 247.381,Z 418.107,A -85,B 0,C 180,E1 -21446.353,E2 -21446.353} C_VEL
LIN {X 0,Y 250.223,Z 424.386,A -85,B 0,C 180,E1 -21447.495,E2 -21447.495} C_VEL
LIN {X 0,Y 246.05,Z 483.615,A -85,B 0,C 180,E1 -21449.113,E2 -21449.113} C_VEL
LIN {X 0,Y 244.094,Z 498.328,A -85,B 0,C 180,E1 -21449.793,E2 -21449.793} C_VEL
LIN {X 0,Y 241.336,Z 512.768,A -85,B 0,C 180,E1 -21450.791,E2 -21450.791} C_VEL
LIN {X 0,Y 238.194,Z 525.458,A -85,B 0,C 180,E1 -21451.983,E2 -21451.983} C_VEL
LIN {X 0,Y 234.627,Z 537.174,A -85,B 0,C 180,E1 -21453.391,E2 -21453.391} C_VEL
LIN {X 0,Y 230.591,Z 548.342,A -85,B 0,C 180,E1 -21455.073,E2 -21455.073} C_VEL
LIN {X 0,Y 225.974,Z 559.403,A -85,B 0,C 180,E1 -21457.163,E2 -21457.163} C_VEL
LIN {X 0,Y 221.288,Z 569.427,A -85,B 0,C 180,E1 -21459.562,E2 -21459.562} C_VEL
LIN {X 0,Y 216.548,Z 578.569,A -85,B 0,C 180,E1 -21462.325,E2 -21462.325} C_VEL
LIN {X 0,Y 212.199,Z 586.214,A -85,B 0,C 180,E1 -21465.271,E2 -21465.271} C_VEL
LIN {X 0,Y 207.931,Z 593.188,A -85,B 0,C 180,E1 -21468.772,E2 -21468.772} C_VEL
LIN {X 0,Y 204.579,Z 598.345,A -85,B 0,C 180,E1 -21472.196,E2 -21472.196} C_VEL
LIN {X 0,Y 201.647,Z 602.591,A -85,B 0,C 180,E1 -21476.109,E2 -21476.109} C_VEL
LIN {X 0,Y 199.349,Z 605.594,A -85,B 0,C 180,E1 -21480.427,E2 -21480.427} C_VEL
LIN {X 0,Y 197.885,Z 607.059,A -85,B 0,C 180,E1 -21484.776,E2 -21484.776} C_VEL
LIN {X 0,Y 197.139,Z 607.039,A -85,B 0,C 180,E1 -21489.117,E2 -21489.117} C_VEL
LIN {X 0,Y 196.971,Z 605.54,A -85,B 0,C 180,E1 -21493.417,E2 -21493.417} C_VEL
LIN {X 0,Y 197.107,Z 604.251,A -85,B 0,C 180,E1 -21495.549,E2 -21495.549} C_VEL
LIN {X 0,Y 197.721,Z 600.582,A -85,B 0,C 180,E1 -21499.765,E2 -21499.765} C_VEL
LIN {X 0,Y 198.448,Z 597.28,A -85,B 0,C 180,E1 -21502.568,E2 -21502.568} C_VEL
LIN {X 0,Y 199.635,Z 592.157,A -85,B 0,C 180,E1 -21505.964,E2 -21505.964} C_VEL
LIN {X 0,Y 201.337,Z 585.381,A -85,B 0,C 180,E1 -21509.502,E2 -21509.502} C_VEL
LIN {X 0,Y 203.371,Z 578.127,A -85,B 0,C 180,E1 -21512.527,E2 -21512.527} C_VEL
LIN {X 0,Y 205.726,Z 569.703,A -85,B 0,C 180,E1 -21515.392,E2 -21515.392} C_VEL
LIN {X 0,Y 208.454,Z 559.387,A -85,B 0,C 180,E1 -21518.24,E2 -21518.24} C_VEL
LIN {X 0,Y 211.193,Z 548.962,A -85,B 0,C 180,E1 -21520.548,E2 -21520.548} C_VEL
LIN {X 0,Y 213.788,Z 537.674,A -85,B 0,C 180,E1 -21522.581,E2 -21522.581} C_VEL
LIN {X 0,Y 216.368,Z 525.322,A -85,B 0,C 180,E1 -21524.341,E2 -21524.341} C_VEL
LIN {X 0,Y 218.738,Z 511.599,A -85,B 0,C 180,E1 -21525.851,E2 -21525.851} C_VEL
LIN {X 0,Y 220.551,Z 497.258,A -85,B 0,C 180,E1 -21527.025,E2 -21527.025} C_VEL
LIN {X 0,Y 221.907,Z 482.752,A -85,B 0,C 180,E1 -21527.819,E2 -21527.819} C_VEL
LIN {X 0,Y 225.751,Z 405.129,A -85,B 0,C 180,E1 -21530.213,E2 -21530.213} C_VEL
LIN {X 0,Y 223.284,Z 398.232,A -85,B 0,C 180,E1 -21530.88,E2 -21530.88} C_VEL
LIN {X 0,Y 219.029,Z 388.772,A -85,B 0,C 180,E1 -21531.982,E2 -21531.982} C_VEL
LIN {X 0,Y 210.212,Z 372.326,A -85,B 0,C 180,E1 -21534.309,E2 -21534.309} C_VEL
LIN {X 0,Y 203.71,Z 361.705,A -85,B 0,C 180,E1 -21536.118,E2 -21536.118} C_VEL
LIN {X 0,Y 201.682,Z 358.376,A -85,B 0,C 180,E1 -21536.716,E2 -21536.716} C_VEL
LIN {X 0,Y 200.069,Z 355.885,A -85,B 0,C 180,E1 -21537.197,E2 -21537.197} C_VEL
LIN {X 0,Y 199.655,Z 354.24,A -85,B 0,C 180,E1 -21537.375,E2 -21537.375} C_VEL
LIN {X 0,Y 199.665,Z 354.238,A -85,B 0,C 180,E1 -21542.354,E2 -21542.354} C_VEL
LIN {X 0,Y 199.618,Z 354.225,A -85,B 0,C 180,E1 -21546.766,E2 -21546.766} C_VEL
LIN {X 0,Y 199.595,Z 354.247,A -85,B 0,C 180,E1 -21549.333,E2 -21549.333} C_VEL
LIN {X 0,Y 199.567,Z 354.238,A -85,B 0,C 180,E1 -21552.309,E2 -21552.309} C_VEL
LIN {X 0,Y 199.577,Z 354.223,A -85,B 0,C 180,E1 -21555.229,E2 -21555.229} C_VEL
LIN {X 0,Y 199.571,Z 354.246,A -85,B 0,C 180,E1 -21558.004,E2 -21558.004} C_VEL
LIN {X 0,Y 199.598,Z 354.237,A -85,B 0,C 180,E1 -21560.775,E2 -21560.775} C_VEL
LIN {X 0,Y 199.612,Z 354.219,A -85,B 0,C 180,E1 -21565.714,E2 -21565.714} C_VEL
LIN {X 0,Y 199.688,Z 354.232,A -85,B 0,C 180,E1 -21568.136,E2 -21568.136} C_VEL
LIN {X 0,Y 199.637,Z 354.234,A -85,B 0,C 180,E1 -21572.765,E2 -21572.765} C_VEL
LIN {X 0,Y 199.674,Z 354.232,A -85,B 0,C 180,E1 -21577.222,E2 -21577.222} C_VEL
LIN {X 0,Y 199.749,Z 354.228,A -85,B 0,C 180,E1 -21581.804,E2 -21581.804} C_VEL
LIN {X 0,Y 199.774,Z 354.192,A -85,B 0,C 180,E1 -21585.745,E2 -21585.745} C_VEL
LIN {X 0,Y 200.028,Z 354.171,A -85,B 0,C 180,E1 -21589.883,E2 -21589.883} C_VEL
LIN {X 0,Y 200.009,Z 354.196,A -85,B 0,C 180,E1 -21593.95,E2 -21593.95} C_VEL
LIN {X 0,Y 200.297,Z 354.128,A -85,B 0,C 180,E1 -21597.99,E2 -21597.99} C_VEL
LIN {X 0,Y 200.472,Z 354.098,A -85,B 0,C 180,E1 -21600.001,E2 -21600.001} C_VEL
LIN {X 0,Y 200.003,Z 354.192,A -85,B 0,C 180,E1 -21604.031,E2 -21604.031} C_VEL
LIN {X 0,Y 200.084,Z 354.178,A -85,B 0,C 180,E1 -21608.078,E2 -21608.078} C_VEL
LIN {X 0,Y 199.879,Z 354.21,A -85,B 0,C 180,E1 -21612.18,E2 -21612.18} C_VEL
LIN {X 0,Y 199.81,Z 354.221,A -85,B 0,C 180,E1 -21616.344,E2 -21616.344} C_VEL
LIN {X 0,Y 199.706,Z 354.226,A -85,B 0,C 180,E1 -21620.605,E2 -21620.605} C_VEL
LIN {X 0,Y 199.679,Z 354.226,A -85,B 0,C 180,E1 -21624.984,E2 -21624.984} C_VEL
LIN {X 0,Y 199.67,Z 354.23,A -85,B 0,C 180,E1 -21629.524,E2 -21629.524} C_VEL
LIN {X 0,Y 199.677,Z 354.235,A -85,B 0,C 180,E1 -21632.355,E2 -21632.355} C_VEL
LIN {X 0,Y 199.628,Z 354.234,A -85,B 0,C 180,E1 -21636.763,E2 -21636.763} C_VEL
LIN {X 0,Y 199.613,Z 354.234,A -85,B 0,C 180,E1 -21639.328,E2 -21639.328} C_VEL
LIN {X 0,Y 199.601,Z 354.388,A -85,B 0,C 180,E1 -21642.706,E2 -21642.706} C_VEL
LIN {X 0,Y 200.598,Z 357.812,A -85,B 0,C 180,E1 -21644.484,E2 -21644.484} C_VEL
LIN {X 0,Y 207.984,Z 372.014,A -85,B 0,C 180,E1 -21646.699,E2 -21646.699} C_VEL
LIN {X 0,Y 213.138,Z 382.897,A -85,B 0,C 180,E1 -21648.172,E2 -21648.172} C_VEL
LIN {X 0,Y 215.036,Z 388.066,A -85,B 0,C 180,E1 -21648.738,E2 -21648.738} C_VEL
LIN {X 0,Y 216.177,Z 393.645,A -85,B 0,C 180,E1 -21649.172,E2 -21649.172} C_VEL
LIN {X 0,Y 217.901,Z 413.2,A -85,B 0,C 180,E1 -21650.264,E2 -21650.264} C_VEL
LIN {X 0,Y 219.016,Z 425.028,A -85,B 0,C 180,E1 -21650.92,E2 -21650.92} C_VEL
LIN {X 0,Y 215.435,Z 496.22,A -85,B 0,C 180,E1 -21653.169,E2 -21653.169} C_VEL
LIN {X 0,Y 213.936,Z 511.018,A -85,B 0,C 180,E1 -21653.966,E2 -21653.966} C_VEL
LIN {X 0,Y 211.854,Z 525.112,A -85,B 0,C 180,E1 -21655.091,E2 -21655.091} C_VEL
LIN {X 0,Y 209.212,Z 539.11,A -85,B 0,C 180,E1 -21656.626,E2 -21656.626} C_VEL
LIN {X 0,Y 206.508,Z 551.177,A -85,B 0,C 180,E1 -21658.354,E2 -21658.354} C_VEL
LIN {X 0,Y 204.165,Z 560.744,A -85,B 0,C 180,E1 -21660.055,E2 -21660.055} C_VEL
LIN {X 0,Y 201.213,Z 571.679,A -85,B 0,C 180,E1 -21662.43,E2 -21662.43} C_VEL
LIN {X 0,Y 198.566,Z 580.818,A -85,B 0,C 180,E1 -21664.865,E2 -21664.865} C_VEL
LIN {X 0,Y 195.991,Z 590.005,A -85,B 0,C 180,E1 -21667.88,E2 -21667.88} C_VEL
LIN {X 0,Y 193.637,Z 598.771,A -85,B 0,C 180,E1 -21671.482,E2 -21671.482} C_VEL
LIN {X 0,Y 191.942,Z 605.816,A -85,B 0,C 180,E1 -21675.147,E2 -21675.147} C_VEL
LIN {X 0,Y 190.927,Z 610.657,A -85,B 0,C 180,E1 -21678.318,E2 -21678.318} C_VEL
LIN {X 0,Y 190.465,Z 614.566,A -85,B 0,C 180,E1 -21681.51,E2 -21681.51} C_VEL
LIN {X 0,Y 190.245,Z 618.344,A -85,B 0,C 180,E1 -21685.761,E2 -21685.761} C_VEL
LIN {X 0,Y 190.427,Z 620.667,A -85,B 0,C 180,E1 -21689.998,E2 -21689.998} C_VEL
LIN {X 0,Y 190.164,Z 621.578,A -85,B 0,C 180,E1 -21694.237,E2 -21694.237} C_VEL
LIN {X 0,Y 190.44,Z 621.168,A -85,B 0,C 180,E1 -21698.487,E2 -21698.487} C_VEL
LIN {X 0,Y 191.351,Z 619.452,A -85,B 0,C 180,E1 -21702.729,E2 -21702.729} C_VEL
LIN {X 0,Y 193.295,Z 616.409,A -85,B 0,C 180,E1 -21706.908,E2 -21706.908} C_VEL
LIN {X 0,Y 195.998,Z 611.957,A -85,B 0,C 180,E1 -21711.011,E2 -21711.011} C_VEL
LIN {X 0,Y 199.796,Z 605.976,A -85,B 0,C 180,E1 -21714.966,E2 -21714.966} C_VEL
LIN {X 0,Y 203.925,Z 599.296,A -85,B 0,C 180,E1 -21718.284,E2 -21718.284} C_VEL
LIN {X 0,Y 208.82,Z 591.052,A -85,B 0,C 180,E1 -21721.442,E2 -21721.442} C_VEL
LIN {X 0,Y 213.539,Z 582.509,A -85,B 0,C 180,E1 -21724.019,E2 -21724.019} C_VEL
LIN {X 0,Y 218.803,Z 571.787,A -85,B 0,C 180,E1 -21726.581,E2 -21726.581} C_VEL
LIN {X 0,Y 223.162,Z 561.917,A -85,B 0,C 180,E1 -21728.459,E2 -21728.459} C_VEL
LIN {X 0,Y 227.582,Z 550.766,A -85,B 0,C 180,E1 -21730.137,E2 -21730.137} C_VEL
LIN {X 0,Y 231.155,Z 540.355,A -85,B 0,C 180,E1 -21731.395,E2 -21731.395} C_VEL
LIN {X 0,Y 234.938,Z 527.441,A -85,B 0,C 180,E1 -21732.592,E2 -21732.592} C_VEL
LIN {X 0,Y 237.924,Z 514.247,A -85,B 0,C 180,E1 -21733.519,E2 -21733.519} C_VEL
LIN {X 0,Y 240.278,Z 499.925,A -85,B 0,C 180,E1 -21734.218,E2 -21734.218} C_VEL
LIN {X 0,Y 241.858,Z 482.441,A -85,B 0,C 180,E1 -21734.774,E2 -21734.774} C_VEL
LIN {X 0,Y 245.077,Z 435.94,A -85,B 0,C 180,E1 -21736.047,E2 -21736.047} C_VEL
LIN {X 0,Y 239.607,Z 423.209,A -85,B 0,C 180,E1 -21738.461,E2 -21738.461} C_VEL
LIN {X 0,Y 234.334,Z 412.604,A -85,B 0,C 180,E1 -21740.963,E2 -21740.963} C_VEL
LIN {X 0,Y 228.95,Z 402.879,A -85,B 0,C 180,E1 -21743.833,E2 -21743.833} C_VEL
LIN {X 0,Y 225.22,Z 396.658,A -85,B 0,C 180,E1 -21746.038,E2 -21746.038} C_VEL
LIN {X 0,Y 222.453,Z 392.26,A -85,B 0,C 180,E1 -21747.826,E2 -21747.826} C_VEL
LIN {X 0,Y 218.913,Z 386.817,A -85,B 0,C 180,E1 -21750.372,E2 -21750.372} C_VEL
LIN {X 0,Y 215.33,Z 381.46,A -85,B 0,C 180,E1 -21753.44,E2 -21753.44} C_VEL
LIN {X 0,Y 211.484,Z 376.537,A -85,B 0,C 180,E1 -21757.448,E2 -21757.448} C_VEL
LIN {X 0,Y 209.787,Z 373.807,A -85,B 0,C 180,E1 -21759.78,E2 -21759.78} C_VEL
LIN {X 0,Y 208.758,Z 372.846,A -85,B 0,C 180,E1 -21761.347,E2 -21761.347} C_VEL
LIN {X 0,Y 205.935,Z 369.487,A -85,B 0,C 180,E1 -21770.175,E2 -21770.175} C_VEL
LIN {X 0,Y 205.954,Z 369.499,A -85,B 0,C 180,E1 -21772.647,E2 -21772.647} C_VEL
LIN {X 0,Y 208.587,Z 372.359,A -85,B 0,C 180,E1 -21780.844,E2 -21780.844} C_VEL
LIN {X 0,Y 210.035,Z 373.31,A -85,B 0,C 180,E1 -21783.016,E2 -21783.016} C_VEL
LIN {X 0,Y 211.66,Z 376.393,A -85,B 0,C 180,E1 -21785.274,E2 -21785.274} C_VEL
LIN {X 0,Y 214.529,Z 379.045,A -85,B 0,C 180,E1 -21788.214,E2 -21788.214} C_VEL
LIN {X 0,Y 216.529,Z 382.258,A -85,B 0,C 180,E1 -21790.106,E2 -21790.106} C_VEL
LIN {X 0,Y 218.551,Z 384.315,A -85,B 0,C 180,E1 -21791.72,E2 -21791.72} C_VEL
LIN {X 0,Y 221.217,Z 387.995,A -85,B 0,C 180,E1 -21793.703,E2 -21793.703} C_VEL
LIN {X 0,Y 222.59,Z 389.843,A -85,B 0,C 180,E1 -21794.63,E2 -21794.63} C_VEL
LIN {X 0,Y 225.994,Z 394.402,A -85,B 0,C 180,E1 -21796.754,E2 -21796.754} C_VEL
LIN {X 0,Y 229.524,Z 399.445,A -85,B 0,C 180,E1 -21798.765,E2 -21798.765} C_VEL
LIN {X 0,Y 234.34,Z 406.578,A -85,B 0,C 180,E1 -21801.246,E2 -21801.246} C_VEL
LIN {X 0,Y 240.494,Z 416.585,A -85,B 0,C 180,E1 -21804.058,E2 -21804.058} C_VEL
LIN {X 0,Y 244.819,Z 425.056,A -85,B 0,C 180,E1 -21805.901,E2 -21805.901} C_VEL
LIN {X 0,Y 245.696,Z 427.041,A -85,B 0,C 180,E1 -21806.271,E2 -21806.271} C_VEL
LIN {X 0,Y 241.44,Z 484.612,A -85,B 0,C 180,E1 -21807.859,E2 -21807.859} C_VEL
LIN {X 0,Y 239.397,Z 499.253,A -85,B 0,C 180,E1 -21808.552,E2 -21808.552} C_VEL
LIN {X 0,Y 236.688,Z 512.889,A -85,B 0,C 180,E1 -21809.501,E2 -21809.501} C_VEL
LIN {X 0,Y 233.427,Z 525.581,A -85,B 0,C 180,E1 -21810.691,E2 -21810.691} C_VEL
LIN {X 0,Y 229.458,Z 538.104,A -85,B 0,C 180,E1 -21812.212,E2 -21812.212} C_VEL
LIN {X 0,Y 225.311,Z 549.081,A -85,B 0,C 180,E1 -21813.897,E2 -21813.897} C_VEL
LIN {X 0,Y 220.482,Z 560.122,A -85,B 0,C 180,E1 -21816.02,E2 -21816.02} C_VEL
LIN {X 0,Y 215.51,Z 570.235,A -85,B 0,C 180,E1 -21818.498,E2 -21818.498} C_VEL
LIN {X 0,Y 210.541,Z 579.274,A -85,B 0,C 180,E1 -21821.322,E2 -21821.322} C_VEL
LIN {X 0,Y 206.077,Z 586.678,A -85,B 0,C 180,E1 -21824.263,E2 -21824.263} C_VEL
LIN {X 0,Y 201.974,Z 593.032,A -85,B 0,C 180,E1 -21827.498,E2 -21827.498} C_VEL
LIN {X 0,Y 198.089,Z 598.658,A -85,B 0,C 180,E1 -21831.309,E2 -21831.309} C_VEL
LIN {X 0,Y 195.288,Z 602.478,A -85,B 0,C 180,E1 -21834.847,E2 -21834.847} C_VEL
LIN {X 0,Y 192.706,Z 605.63,A -85,B 0,C 180,E1 -21839.3,E2 -21839.3} C_VEL
LIN {X 0,Y 191.027,Z 607.237,A -85,B 0,C 180,E1 -21843.804,E2 -21843.804} C_VEL
LIN {X 0,Y 190.148,Z 607.365,A -85,B 0,C 180,E1 -21848.311,E2 -21848.311} C_VEL
LIN {X 0,Y 189.856,Z 606.049,A -85,B 0,C 180,E1 -21852.776,E2 -21852.776} C_VEL
LIN {X 0,Y 189.993,Z 604.835,A -85,B 0,C 180,E1 -21854.995,E2 -21854.995} C_VEL
LIN {X 0,Y 190.558,Z 601.304,A -85,B 0,C 180,E1 -21859.376,E2 -21859.376} C_VEL
LIN {X 0,Y 191.346,Z 597.707,A -85,B 0,C 180,E1 -21862.602,E2 -21862.602} C_VEL
LIN {X 0,Y 192.439,Z 593.101,A -85,B 0,C 180,E1 -21865.813,E2 -21865.813} C_VEL
LIN {X 0,Y 194.166,Z 586.497,A -85,B 0,C 180,E1 -21869.483,E2 -21869.483} C_VEL
LIN {X 0,Y 196.21,Z 579.418,A -85,B 0,C 180,E1 -21872.619,E2 -21872.619} C_VEL
LIN {X 0,Y 198.65,Z 571.106,A -85,B 0,C 180,E1 -21875.616,E2 -21875.616} C_VEL
LIN {X 0,Y 201.388,Z 561.172,A -85,B 0,C 180,E1 -21878.531,E2 -21878.531} C_VEL
LIN {X 0,Y 204.463,Z 549.97,A -85,B 0,C 180,E1 -21881.15,E2 -21881.15} C_VEL
LIN {X 0,Y 207.156,Z 538.841,A -85,B 0,C 180,E1 -21883.24,E2 -21883.24} C_VEL
LIN {X 0,Y 209.818,Z 526.717,A -85,B 0,C 180,E1 -21885.047,E2 -21885.047} C_VEL
LIN {X 0,Y 212.223,Z 513.332,A -85,B 0,C 180,E1 -21886.598,E2 -21886.598} C_VEL
LIN {X 0,Y 214.191,Z 499.152,A -85,B 0,C 180,E1 -21887.817,E2 -21887.817} C_VEL
LIN {X 0,Y 215.589,Z 485.229,A -85,B 0,C 180,E1 -21888.642,E2 -21888.642} C_VEL
LIN {X 0,Y 216.855,Z 464.215,A -85,B 0,C 180,E1 -21889.37,E2 -21889.37} C_VEL
LIN {X 0,Y 219.643,Z 406.276,A -85,B 0,C 180,E1 -21891.179,E2 -21891.179} C_VEL
LIN {X 0,Y 215.441,Z 396.015,A -85,B 0,C 180,E1 -21892.332,E2 -21892.332} C_VEL
LIN {X 0,Y 207.102,Z 379.802,A -85,B 0,C 180,E1 -21894.611,E2 -21894.611} C_VEL
LIN {X 0,Y 199.406,Z 366.729,A -85,B 0,C 180,E1 -21896.844,E2 -21896.844} C_VEL
LIN {X 0,Y 194.583,Z 359.197,A -85,B 0,C 180,E1 -21898.337,E2 -21898.337} C_VEL
LIN {X 0,Y 192.942,Z 356.599,A -85,B 0,C 180,E1 -21898.872,E2 -21898.872} C_VEL
LIN {X 0,Y 192.584,Z 355.119,A -85,B 0,C 180,E1 -21899.063,E2 -21899.063} C_VEL
LIN {X 0,Y 192.595,Z 355.123,A -85,B 0,C 180,E1 -21903.188,E2 -21903.188} C_VEL
LIN {X 0,Y 192.542,Z 355.116,A -85,B 0,C 180,E1 -21908.356,E2 -21908.356} C_VEL
LIN {X 0,Y 192.485,Z 355.109,A -85,B 0,C 180,E1 -21913.095,E2 -21913.095} C_VEL
LIN {X 0,Y 192.485,Z 355.12,A -85,B 0,C 180,E1 -21916.909,E2 -21916.909} C_VEL
LIN {X 0,Y 192.542,Z 355.104,A -85,B 0,C 180,E1 -21921.647,E2 -21921.647} C_VEL
LIN {X 0,Y 192.597,Z 355.104,A -85,B 0,C 180,E1 -21926.815,E2 -21926.815} C_VEL
LIN {X 0,Y 192.621,Z 355.108,A -85,B 0,C 180,E1 -21931.686,E2 -21931.686} C_VEL
LIN {X 0,Y 192.665,Z 355.109,A -85,B 0,C 180,E1 -21936.344,E2 -21936.344} C_VEL
LIN {X 0,Y 192.698,Z 355.105,A -85,B 0,C 180,E1 -21941.493,E2 -21941.493} C_VEL
LIN {X 0,Y 192.778,Z 355.05,A -85,B 0,C 180,E1 -21947.366,E2 -21947.366} C_VEL
LIN {X 0,Y 193.026,Z 355.057,A -85,B 0,C 180,E1 -21951.627,E2 -21951.627} C_VEL
LIN {X 0,Y 193.241,Z 355.006,A -85,B 0,C 180,E1 -21957.916,E2 -21957.916} C_VEL
LIN {X 0,Y 193.436,Z 354.972,A -85,B 0,C 180,E1 -21960.001,E2 -21960.001} C_VEL
LIN {X 0,Y 192.951,Z 355.071,A -85,B 0,C 180,E1 -21964.178,E2 -21964.178} C_VEL
LIN {X 0,Y 193.034,Z 355.055,A -85,B 0,C 180,E1 -21968.375,E2 -21968.375} C_VEL
LIN {X 0,Y 192.807,Z 355.089,A -85,B 0,C 180,E1 -21972.634,E2 -21972.634} C_VEL
LIN {X 0,Y 192.764,Z 355.098,A -85,B 0,C 180,E1 -21976.959,E2 -21976.959} C_VEL
LIN {X 0,Y 192.643,Z 355.109,A -85,B 0,C 180,E1 -21981.397,E2 -21981.397} C_VEL
LIN {X 0,Y 192.67,Z 355.101,A -85,B 0,C 180,E1 -21984.224,E2 -21984.224} C_VEL
LIN {X 0,Y 192.65,Z 355.106,A -85,B 0,C 180,E1 -21988.889,E2 -21988.889} C_VEL
LIN {X 0,Y 192.602,Z 355.113,A -85,B 0,C 180,E1 -21993.186,E2 -21993.186} C_VEL
LIN {X 0,Y 192.556,Z 355.107,A -85,B 0,C 180,E1 -21998.351,E2 -21998.351} C_VEL
LIN {X 0,Y 192.535,Z 355.161,A -85,B 0,C 180,E1 -22001.434,E2 -22001.434} C_VEL
LIN {X 0,Y 193.284,Z 357.744,A -85,B 0,C 180,E1 -22002.744,E2 -22002.744} C_VEL
LIN {X 0,Y 195.701,Z 362.039,A -85,B 0,C 180,E1 -22003.543,E2 -22003.543} C_VEL
LIN {X 0,Y 202.728,Z 375.394,A -85,B 0,C 180,E1 -22005.752,E2 -22005.752} C_VEL
LIN {X 0,Y 209.775,Z 390.813,A -85,B 0,C 180,E1 -22007.858,E2 -22007.858} C_VEL
LIN {X 0,Y 216.126,Z 407.251,A -85,B 0,C 180,E1 -22009.715,E2 -22009.715} C_VEL
LIN {X 0,Y 217.793,Z 412.381,A -85,B 0,C 180,E1 -22010.213,E2 -22010.213} C_VEL
LIN {X 0,Y 217.901,Z 413.2,A -85,B 0,C 180,E1 -22010.264,E2 -22010.264} C_VEL
LIN {X 0,Y 218.015,Z 417.069,A -85,B 0,C 180,E1 -22010.437,E2 -22010.437} C_VEL
LIN {X 0,Y 217.557,Z 420.972,A -85,B 0,C 180,E1 -22010.514,E2 -22010.514} C_VEL
LIN {X 0,Y 215.619,Z 428.703,A -85,B 0,C 180,E1 -22010.489,E2 -22010.489} C_VEL
LIN {X 0,Y 213.347,Z 436.482,A -85,B 0,C 180,E1 -22010.407,E2 -22010.407} C_VEL
LIN {X 0,Y 212.219,Z 442.406,A -85,B 0,C 180,E1 -22010.449,E2 -22010.449} C_VEL
LIN {X 0,Y 212.065,Z 444.4,A -85,B 0,C 180,E1 -22010.503,E2 -22010.503} C_VEL
LIN {X 0,Y 209.319,Z 496.538,A -85,B 0,C 180,E1 -22012.209,E2 -22012.209} C_VEL
LIN {X 0,Y 207.76,Z 511.12,A -85,B 0,C 180,E1 -22013.021,E2 -22013.021} C_VEL
LIN {X 0,Y 205.615,Z 525.121,A -85,B 0,C 180,E1 -22014.171,E2 -22014.171} C_VEL
LIN {X 0,Y 202.884,Z 539.06,A -85,B 0,C 180,E1 -22015.741,E2 -22015.741} C_VEL
LIN {X 0,Y 200.025,Z 551.267,A -85,B 0,C 180,E1 -22017.539,E2 -22017.539} C_VEL
LIN {X 0,Y 197.656,Z 560.623,A -85,B 0,C 180,E1 -22019.259,E2 -22019.259} C_VEL
LIN {X 0,Y 194.871,Z 570.539,A -85,B 0,C 180,E1 -22021.452,E2 -22021.452} C_VEL
LIN {X 0,Y 192.064,Z 579.819,A -85,B 0,C 180,E1 -22023.951,E2 -22023.951} C_VEL
LIN {X 0,Y 189.35,Z 589.131,A -85,B 0,C 180,E1 -22027.061,E2 -22027.061} C_VEL
LIN {X 0,Y 186.798,Z 597.999,A -85,B 0,C 180,E1 -22030.778,E2 -22030.778} C_VEL
LIN {X 0,Y 185.014,Z 605.143,A -85,B 0,C 180,E1 -22034.577,E2 -22034.577} C_VEL
LIN {X 0,Y 183.924,Z 610.071,A -85,B 0,C 180,E1 -22037.866,E2 -22037.866} C_VEL
LIN {X 0,Y 183.406,Z 614.058,A -85,B 0,C 180,E1 -22041.181,E2 -22041.181} C_VEL
LIN {X 0,Y 183.157,Z 617.915,A -85,B 0,C 180,E1 -22045.597,E2 -22045.597} C_VEL
LIN {X 0,Y 183.343,Z 620.31,A -85,B 0,C 180,E1 -22049.998,E2 -22049.998} C_VEL
LIN {X 0,Y 183.076,Z 621.29,A -85,B 0,C 180,E1 -22054.401,E2 -22054.401} C_VEL
LIN {X 0,Y 183.389,Z 620.949,A -85,B 0,C 180,E1 -22058.816,E2 -22058.816} C_VEL
LIN {X 0,Y 184.376,Z 619.303,A -85,B 0,C 180,E1 -22063.219,E2 -22063.219} C_VEL
LIN {X 0,Y 186.486,Z 616.333,A -85,B 0,C 180,E1 -22067.545,E2 -22067.545} C_VEL
LIN {X 0,Y 189.462,Z 611.74,A -85,B 0,C 180,E1 -22071.971,E2 -22071.971} C_VEL
LIN {X 0,Y 193.369,Z 606.077,A -85,B 0,C 180,E1 -22075.855,E2 -22075.855} C_VEL
LIN {X 0,Y 197.702,Z 599.51,A -85,B 0,C 180,E1 -22079.259,E2 -22079.259} C_VEL
LIN {X 0,Y 202.812,Z 591.415,A -85,B 0,C 180,E1 -22082.485,E2 -22082.485} C_VEL
LIN {X 0,Y 207.71,Z 582.985,A -85,B 0,C 180,E1 -22085.111,E2 -22085.111} C_VEL
LIN {X 0,Y 213.056,Z 572.708,A -85,B 0,C 180,E1 -22087.656,E2 -22087.656} C_VEL
LIN {X 0,Y 218.204,Z 561.599,A -85,B 0,C 180,E1 -22089.8,E2 -22089.8} C_VEL
LIN {X 0,Y 222.756,Z 550.445,A -85,B 0,C 180,E1 -22091.492,E2 -22091.492} C_VEL
LIN {X 0,Y 227.019,Z 538.314,A -85,B 0,C 180,E1 -22092.925,E2 -22092.925} C_VEL
LIN {X 0,Y 230.926,Z 524.873,A -85,B 0,C 180,E1 -22094.118,E2 -22094.118} C_VEL
LIN {X 0,Y 233.772,Z 512.358,A -85,B 0,C 180,E1 -22094.947,E2 -22094.947} C_VEL
LIN {X 0,Y 236.196,Z 497.14,A -85,B 0,C 180,E1 -22095.654,E2 -22095.654} C_VEL
LIN {X 0,Y 238.15,Z 473.957,A -85,B 0,C 180,E1 -22096.327,E2 -22096.327} C_VEL
LIN {X 0,Y 240.619,Z 438.567,A -85,B 0,C 180,E1 -22097.326,E2 -22097.326} C_VEL
LIN {X 0,Y 235.662,Z 426.917,A -85,B 0,C 180,E1 -22099.652,E2 -22099.652} C_VEL
LIN {X 0,Y 231.01,Z 417.389,A -85,B 0,C 180,E1 -22102.022,E2 -22102.022} C_VEL
LIN {X 0,Y 226.326,Z 408.584,A -85,B 0,C 180,E1 -22104.667,E2 -22104.667} C_VEL
LIN {X 0,Y 222.531,Z 402.082,A -85,B 0,C 180,E1 -22107.036,E2 -22107.036} C_VEL
LIN {X 0,Y 220.249,Z 398.351,A -85,B 0,C 180,E1 -22108.593,E2 -22108.593} C_VEL
LIN {X 0,Y 217.021,Z 393.157,A -85,B 0,C 180,E1 -22111.066,E2 -22111.066} C_VEL
LIN {X 0,Y 213.259,Z 387.426,A -85,B 0,C 180,E1 -22114.485,E2 -22114.485} C_VEL
LIN {X 0,Y 208.647,Z 380.717,A -85,B 0,C 180,E1 -22120.094,E2 -22120.094} C_VEL
LIN {X 0,Y 207.681,Z 379.778,A -85,B 0,C 180,E1 -22121.649,E2 -22121.649} C_VEL
LIN {X 0,Y 205.043,Z 376.58,A -85,B 0,C 180,E1 -22130.131,E2 -22130.131} C_VEL
LIN {X 0,Y 205.059,Z 376.566,A -85,B 0,C 180,E1 -22132.615,E2 -22132.615} C_VEL
LIN {X 0,Y 207.485,Z 379.28,A -85,B 0,C 180,E1 -22140.485,E2 -22140.485} C_VEL
LIN {X 0,Y 208.842,Z 380.373,A -85,B 0,C 180,E1 -22142.667,E2 -22142.667} C_VEL
LIN {X 0,Y 210.652,Z 383.509,A -85,B 0,C 180,E1 -22145.184,E2 -22145.184} C_VEL
LIN {X 0,Y 212.98,Z 385.728,A -85,B 0,C 180,E1 -22147.644,E2 -22147.644} C_VEL
LIN {X 0,Y 215.316,Z 389.327,A -85,B 0,C 180,E1 -22149.907,E2 -22149.907} C_VEL
LIN {X 0,Y 216.894,Z 391.038,A -85,B 0,C 180,E1 -22151.21,E2 -22151.21} C_VEL
LIN {X 0,Y 219.686,Z 394.83,A -85,B 0,C 180,E1 -22153.357,E2 -22153.357} C_VEL
LIN {X 0,Y 224.34,Z 401.436,A -85,B 0,C 180,E1 -22156.423,E2 -22156.423} C_VEL
LIN {X 0,Y 228.815,Z 407.986,A -85,B 0,C 180,E1 -22159.001,E2 -22159.001} C_VEL
LIN {X 0,Y 233.739,Z 415.893,A -85,B 0,C 180,E1 -22161.557,E2 -22161.557} C_VEL
LIN {X 0,Y 238.742,Z 424.555,A -85,B 0,C 180,E1 -22163.878,E2 -22163.878} C_VEL
LIN {X 0,Y 241.192,Z 429.685,A -85,B 0,C 180,E1 -22164.971,E2 -22164.971} C_VEL
LIN {X 0,Y 237.164,Z 483.947,A -85,B 0,C 180,E1 -22166.494,E2 -22166.494} C_VEL
LIN {X 0,Y 235.192,Z 498.112,A -85,B 0,C 180,E1 -22167.141,E2 -22167.141} C_VEL
LIN {X 0,Y 232.433,Z 511.785,A -85,B 0,C 180,E1 -22168.055,E2 -22168.055} C_VEL
LIN {X 0,Y 228.983,Z 524.931,A -85,B 0,C 180,E1 -22169.256,E2 -22169.256} C_VEL
LIN {X 0,Y 224.947,Z 537.52,A -85,B 0,C 180,E1 -22170.779,E2 -22170.779} C_VEL
LIN {X 0,Y 220.232,Z 549.547,A -85,B 0,C 180,E1 -22172.616,E2 -22172.616} C_VEL
LIN {X 0,Y 215.081,Z 560.84,A -85,B 0,C 180,E1 -22174.82,E2 -22174.82} C_VEL
LIN {X 0,Y 209.684,Z 571.265,A -85,B 0,C 180,E1 -22177.449,E2 -22177.449} C_VEL
LIN {X 0,Y 204.729,Z 579.825,A -85,B 0,C 180,E1 -22180.203,E2 -22180.203} C_VEL
LIN {X 0,Y 200.04,Z 587.178,A -85,B 0,C 180,E1 -22183.2,E2 -22183.2} C_VEL
LIN {X 0,Y 195.287,Z 594.047,A -85,B 0,C 180,E1 -22186.864,E2 -22186.864} C_VEL
LIN {X 0,Y 191.708,Z 598.95,A -85,B 0,C 180,E1 -22190.34,E2 -22190.34} C_VEL
LIN {X 0,Y 189.035,Z 602.331,A -85,B 0,C 180,E1 -22193.501,E2 -22193.501} C_VEL
LIN {X 0,Y 187.474,Z 604.213,A -85,B 0,C 180,E1 -22195.786,E2 -22195.786} C_VEL
LIN {X 0,Y 185.097,Z 606.729,A -85,B 0,C 180,E1 -22200.425,E2 -22200.425} C_VEL
LIN {X 0,Y 183.582,Z 607.732,A -85,B 0,C 180,E1 -22205.098,E2 -22205.098} C_VEL
LIN {X 0,Y 183.172,Z 607.681,A -85,B 0,C 180,E1 -22207.44,E2 -22207.44} C_VEL
LIN {X 0,Y 182.759,Z 606.504,A -85,B 0,C 180,E1 -22212.085,E2 -22212.085} C_VEL
LIN {X 0,Y 182.873,Z 605.374,A -85,B 0,C 180,E1 -22214.396,E2 -22214.396} C_VEL
LIN {X 0,Y 183.356,Z 602.029,A -85,B 0,C 180,E1 -22218.953,E2 -22218.953} C_VEL
LIN {X 0,Y 184.24,Z 598.116,A -85,B 0,C 180,E1 -22222.648,E2 -22222.648} C_VEL
LIN {X 0,Y 185.684,Z 592.386,A -85,B 0,C 180,E1 -22226.747,E2 -22226.747} C_VEL
LIN {X 0,Y 187.576,Z 585.514,A -85,B 0,C 180,E1 -22230.539,E2 -22230.539} C_VEL
LIN {X 0,Y 189.807,Z 578.319,A -85,B 0,C 180,E1 -22233.717,E2 -22233.717} C_VEL
LIN {X 0,Y 192.356,Z 569.687,A -85,B 0,C 180,E1 -22236.821,E2 -22236.821} C_VEL
LIN {X 0,Y 195.382,Z 559.214,A -85,B 0,C 180,E1 -22239.84,E2 -22239.84} C_VEL
LIN {X 0,Y 198.361,Z 548.646,A -85,B 0,C 180,E1 -22242.276,E2 -22242.276} C_VEL
LIN {X 0,Y 201.236,Z 537.159,A -85,B 0,C 180,E1 -22244.41,E2 -22244.41} C_VEL
LIN {X 0,Y 203.984,Z 524.582,A -85,B 0,C 180,E1 -22246.258,E2 -22246.258} C_VEL
LIN {X 0,Y 206.351,Z 511.645,A -85,B 0,C 180,E1 -22247.724,E2 -22247.724} C_VEL
LIN {X 0,Y 208.287,Z 497.423,A -85,B 0,C 180,E1 -22248.928,E2 -22248.928} C_VEL
LIN {X 0,Y 209.744,Z 482.555,A -85,B 0,C 180,E1 -22249.766,E2 -22249.766} C_VEL
LIN {X 0,Y 213.742,Z 408.55,A -85,B 0,C 180,E1 -22252.128,E2 -22252.128} C_VEL
LIN {X 0,Y 210.254,Z 399.803,A -85,B 0,C 180,E1 -22253.144,E2 -22253.144} C_VEL
LIN {X 0,Y 202.302,Z 384.134,A -85,B 0,C 180,E1 -22255.414,E2 -22255.414} C_VEL
LIN {X 0,Y 194.961,Z 371.517,A -85,B 0,C 180,E1 -22257.651,E2 -22257.651} C_VEL
LIN {X 0,Y 189.709,Z 363.414,A -85,B 0,C 180,E1 -22259.359,E2 -22259.359} C_VEL
LIN {X 0,Y 187.893,Z 360.463,A -85,B 0,C 180,E1 -22259.988,E2 -22259.988} C_VEL
LIN {X 0,Y 186.09,Z 358.006,A -85,B 0,C 180,E1 -22260.604,E2 -22260.604} C_VEL
LIN {X 0,Y 185.518,Z 356.001,A -85,B 0,C 180,E1 -22260.906,E2 -22260.906} C_VEL
LIN {X 0,Y 185.497,Z 355.996,A -85,B 0,C 180,E1 -22264.635,E2 -22264.635} C_VEL
LIN {X 0,Y 185.5,Z 355.983,A -85,B 0,C 180,E1 -22267.316,E2 -22267.316} C_VEL
LIN {X 0,Y 185.462,Z 356.008,A -85,B 0,C 180,E1 -22270.723,E2 -22270.723} C_VEL
LIN {X 0,Y 185.456,Z 355.986,A -85,B 0,C 180,E1 -22276.058,E2 -22276.058} C_VEL
LIN {X 0,Y 185.457,Z 356.005,A -85,B 0,C 180,E1 -22279.894,E2 -22279.894} C_VEL
LIN {X 0,Y 185.502,Z 355.967,A -85,B 0,C 180,E1 -22282.716,E2 -22282.716} C_VEL
LIN {X 0,Y 185.533,Z 355.994,A -85,B 0,C 180,E1 -22287.974,E2 -22287.974} C_VEL
LIN {X 0,Y 185.55,Z 355.993,A -85,B 0,C 180,E1 -22290.597,E2 -22290.597} C_VEL
LIN {X 0,Y 185.566,Z 355.995,A -85,B 0,C 180,E1 -22295.38,E2 -22295.38} C_VEL
LIN {X 0,Y 185.629,Z 355.986,A -85,B 0,C 180,E1 -22301.18,E2 -22301.18} C_VEL
LIN {X 0,Y 185.702,Z 355.931,A -85,B 0,C 180,E1 -22306.876,E2 -22306.876} C_VEL
LIN {X 0,Y 185.977,Z 355.933,A -85,B 0,C 180,E1 -22311.307,E2 -22311.307} C_VEL
LIN {X 0,Y 186.187,Z 355.884,A -85,B 0,C 180,E1 -22317.837,E2 -22317.837} C_VEL
LIN {X 0,Y 186.4,Z 355.846,A -85,B 0,C 180,E1 -22320.001,E2 -22320.001} C_VEL
LIN {X 0,Y 185.899,Z 355.951,A -85,B 0,C 180,E1 -22324.337,E2 -22324.337} C_VEL
LIN {X 0,Y 185.983,Z 355.934,A -85,B 0,C 180,E1 -22328.695,E2 -22328.695} C_VEL
LIN {X 0,Y 185.734,Z 355.968,A -85,B 0,C 180,E1 -22333.123,E2 -22333.123} C_VEL
LIN {X 0,Y 185.696,Z 355.976,A -85,B 0,C 180,E1 -22337.625,E2 -22337.625} C_VEL
LIN {X 0,Y 185.603,Z 355.989,A -85,B 0,C 180,E1 -22342.251,E2 -22342.251} C_VEL
LIN {X 0,Y 185.567,Z 355.992,A -85,B 0,C 180,E1 -22347.032,E2 -22347.032} C_VEL
LIN {X 0,Y 185.583,Z 355.983,A -85,B 0,C 180,E1 -22349.493,E2 -22349.493} C_VEL
LIN {X 0,Y 185.505,Z 356.001,A -85,B 0,C 180,E1 -22354.632,E2 -22354.632} C_VEL
LIN {X 0,Y 185.488,Z 355.992,A -85,B 0,C 180,E1 -22359.394,E2 -22359.394} C_VEL
LIN {X 0,Y 185.492,Z 356.024,A -85,B 0,C 180,E1 -22360.099,E2 -22360.099} C_VEL
LIN {X 0,Y 185.812,Z 357.419,A -85,B 0,C 180,E1 -22360.757,E2 -22360.757} C_VEL
LIN {X 0,Y 192.14,Z 368.485,A -85,B 0,C 180,E1 -22362.986,E2 -22362.986} C_VEL
LIN {X 0,Y 198.384,Z 380.697,A -85,B 0,C 180,E1 -22365.043,E2 -22365.043} C_VEL
LIN {X 0,Y 205.415,Z 396.445,A -85,B 0,C 180,E1 -22367.236,E2 -22367.236} C_VEL
LIN {X 0,Y 211.951,Z 414.122,A -85,B 0,C 180,E1 -22369.242,E2 -22369.242} C_VEL
LIN {X 0,Y 213.031,Z 425.769,A -85,B 0,C 180,E1 -22369.916,E2 -22369.916} C_VEL
LIN {X 0,Y 212.065,Z 444.4,A -85,B 0,C 180,E1 -22370.503,E2 -22370.503} C_VEL
LIN {X 0,Y 211.254,Z 450.238,A -85,B 0,C 180,E1 -22370.599,E2 -22370.599} C_VEL
LIN {X 0,Y 205.459,Z 469.199,A -85,B 0,C 180,E1 -22370.349,E2 -22370.349} C_VEL
LIN {X 0,Y 204.565,Z 475.041,A -85,B 0,C 180,E1 -22370.433,E2 -22370.433} C_VEL
LIN {X 0,Y 203.088,Z 498.314,A -85,B 0,C 180,E1 -22371.258,E2 -22371.258} C_VEL
LIN {X 0,Y 201.428,Z 512.752,A -85,B 0,C 180,E1 -22372.129,E2 -22372.129} C_VEL
LIN {X 0,Y 199.241,Z 526.276,A -85,B 0,C 180,E1 -22373.31,E2 -22373.31} C_VEL
LIN {X 0,Y 196.607,Z 539.01,A -85,B 0,C 180,E1 -22374.8,E2 -22374.8} C_VEL
LIN {X 0,Y 193.558,Z 551.499,A -85,B 0,C 180,E1 -22376.694,E2 -22376.694} C_VEL
LIN {X 0,Y 191.187,Z 560.501,A -85,B 0,C 180,E1 -22378.409,E2 -22378.409} C_VEL
LIN {X 0,Y 187.976,Z 571.382,A -85,B 0,C 180,E1 -22380.917,E2 -22380.917} C_VEL
LIN {X 0,Y 185.117,Z 580.483,A -85,B 0,C 180,E1 -22383.505,E2 -22383.505} C_VEL
LIN {X 0,Y 182.327,Z 589.638,A -85,B 0,C 180,E1 -22386.726,E2 -22386.726} C_VEL
LIN {X 0,Y 179.727,Z 598.372,A -85,B 0,C 180,E1 -22390.585,E2 -22390.585} C_VEL
LIN {X 0,Y 178.113,Z 604.47,A -85,B 0,C 180,E1 -22393.964,E2 -22393.964} C_VEL
LIN {X 0,Y 176.941,Z 609.485,A -85,B 0,C 180,E1 -22397.38,E2 -22397.38} C_VEL
LIN {X 0,Y 176.342,Z 613.525,A -85,B 0,C 180,E1 -22400.825,E2 -22400.825} C_VEL
LIN {X 0,Y 176.143,Z 615.703,A -85,B 0,C 180,E1 -22403.123,E2 -22403.123} C_VEL
LIN {X 0,Y 176.112,Z 618.897,A -85,B 0,C 180,E1 -22407.711,E2 -22407.711} C_VEL
